LIN {X 0,Y 523.917,Z 120.846,A -85,B 0,C 180,E1 -4821.899,E2 -4821.899} C_VEL
LIN {X 0,Y 523.927,Z 120.846,A -85,B 0,C 180,E1 -4824.912,E2 -4824.912} C_VEL
LIN {X 0,Y 523.938,Z 120.844,A -85,B 0,C 180,E1 -4827.68,E2 -4827.68} C_VEL
LIN {X 0,Y 523.939,Z 120.843,A -85,B 0,C 180,E1 -4830.681,E2 -4830.681} C_VEL
LIN {X 0,Y 523.936,Z 120.839,A -85,B 0,C 180,E1 -4833.727,E2 -4833.727} C_VEL
LIN {X 0,Y 523.911,Z 120.845,A -85,B 0,C 180,E1 -4836.27,E2 -4836.27} C_VEL
LIN {X 0,Y 523.949,Z 120.845,A -85,B 0,C 180,E1 -4838.767,E2 -4838.767} C_VEL
LIN {X 0,Y 523.94,Z 120.843,A -85,B 0,C 180,E1 -4841.221,E2 -4841.221} C_VEL
LIN {X 0,Y 523.911,Z 120.843,A -85,B 0,C 180,E1 -4843.638,E2 -4843.638} C_VEL
LIN {X 0,Y 523.917,Z 120.845,A -85,B 0,C 180,E1 -4846.028,E2 -4846.028} C_VEL
LIN {X 0,Y 523.996,Z 120.835,A -85,B 0,C 180,E1 -4849.177,E2 -4849.177} C_VEL
LIN {X 0,Y 523.964,Z 120.844,A -85,B 0,C 180,E1 -4852.292,E2 -4852.292} C_VEL
LIN {X 0,Y 524.035,Z 120.834,A -85,B 0,C 180,E1 -4854.613,E2 -4854.613} C_VEL
LIN {X 0,Y 524.107,Z 120.819,A -85,B 0,C 180,E1 -4857.695,E2 -4857.695} C_VEL
LIN {X 0,Y 524.101,Z 120.817,A -85,B 0,C 180,E1 -4860,E2 -4860} C_VEL
LIN {X 0,Y 524.107,Z 120.825,A -85,B 0,C 180,E1 -4862.306,E2 -4862.306} C_VEL
LIN {X 0,Y 524.004,Z 120.837,A -85,B 0,C 180,E1 -4866.16,E2 -4866.16} C_VEL
LIN {X 0,Y 523.947,Z 120.832,A -85,B 0,C 180,E1 -4869.263,E2 -4869.263} C_VEL
LIN {X 0,Y 523.925,Z 120.843,A -85,B 0,C 180,E1 -4872.394,E2 -4872.394} C_VEL
LIN {X 0,Y 523.924,Z 120.843,A -85,B 0,C 180,E1 -4875.022,E2 -4875.022} C_VEL
LIN {X 0,Y 523.891,Z 120.851,A -85,B 0,C 180,E1 -4877.972,E2 -4877.972} C_VEL
LIN {X 0,Y 523.893,Z 120.847,A -85,B 0,C 180,E1 -4880.414,E2 -4880.414} C_VEL
LIN {X 0,Y 523.887,Z 120.847,A -85,B 0,C 180,E1 -4882.895,E2 -4882.895} C_VEL
LIN {X 0,Y 523.876,Z 120.857,A -85,B 0,C 180,E1 -4885.423,E2 -4885.423} C_VEL
LIN {X 0,Y 523.9,Z 120.841,A -85,B 0,C 180,E1 -4888.003,E2 -4888.003} C_VEL
LIN {X 0,Y 523.902,Z 120.842,A -85,B 0,C 180,E1 -4890.846,E2 -4890.846} C_VEL
LIN {X 0,Y 523.916,Z 120.846,A -85,B 0,C 180,E1 -4893.726,E2 -4893.726} C_VEL
LIN {X 0,Y 523.863,Z 120.849,A -85,B 0,C 180,E1 -4896.394,E2 -4896.394} C_VEL
LIN {X 0,Y 523.904,Z 120.848,A -85,B 0,C 180,E1 -4899.087,E2 -4899.087} C_VEL
LIN {X 0,Y 523.898,Z 120.847,A -85,B 0,C 180,E1 -4902.125,E2 -4902.125} C_VEL
LIN {X 0,Y 523.939,Z 120.837,A -85,B 0,C 180,E1 -4905.311,E2 -4905.311} C_VEL
LIN {X 0,Y 523.883,Z 120.852,A -85,B 0,C 180,E1 -4906.869,E2 -4906.869} C_VEL
LIN {X 0,Y 523.195,Z 120.935,A -85,B 0,C 180,E1 -4907.511,E2 -4907.511} C_VEL
LIN {X 0,Y 520.332,Z 121.296,A -85,B 0,C 180,E1 -4908.552,E2 -4908.552} C_VEL
LIN {X 0,Y 517.938,Z 121.591,A -85,B 0,C 180,E1 -4909.391,E2 -4909.391} C_VEL
LIN {X 0,Y 516.933,Z 121.716,A -85,B 0,C 180,E1 -4910.039,E2 -4910.039} C_VEL
LIN {X 0,Y 516.862,Z 121.727,A -85,B 0,C 180,E1 -4910.258,E2 -4910.258} C_VEL
LIN {X 0,Y 516.858,Z 121.723,A -85,B 0,C 180,E1 -4913.252,E2 -4913.252} C_VEL
LIN {X 0,Y 516.885,Z 121.724,A -85,B 0,C 180,E1 -4916.118,E2 -4916.118} C_VEL
LIN {X 0,Y 516.894,Z 121.721,A -85,B 0,C 180,E1 -4918.936,E2 -4918.936} C_VEL
LIN {X 0,Y 516.853,Z 121.724,A -85,B 0,C 180,E1 -4921.58,E2 -4921.58} C_VEL
LIN {X 0,Y 516.876,Z 121.73,A -85,B 0,C 180,E1 -4924.207,E2 -4924.207} C_VEL
LIN {X 0,Y 516.862,Z 121.725,A -85,B 0,C 180,E1 -4926.776,E2 -4926.776} C_VEL
LIN {X 0,Y 516.943,Z 121.718,A -85,B 0,C 180,E1 -4929.732,E2 -4929.732} C_VEL
LIN {X 0,Y 516.89,Z 121.718,A -85,B 0,C 180,E1 -4932.594,E2 -4932.594} C_VEL
LIN {X 0,Y 516.941,Z 121.714,A -85,B 0,C 180,E1 -4935.03,E2 -4935.03} C_VEL
LIN {X 0,Y 516.973,Z 121.714,A -85,B 0,C 180,E1 -4938.233,E2 -4938.233} C_VEL
LIN {X 0,Y 516.959,Z 121.718,A -85,B 0,C 180,E1 -4941.399,E2 -4941.399} C_VEL
LIN {X 0,Y 517.024,Z 121.796,A -85,B 0,C 180,E1 -4943.952,E2 -4943.952} C_VEL
LIN {X 0,Y 519.184,Z 132.355,A -85,B 0,C 180,E1 -4945.73,E2 -4945.73} C_VEL
LIN {X 0,Y 518.904,Z 142.438,A -85,B 0,C 180,E1 -4947.27,E2 -4947.27} C_VEL
LIN {X 0,Y 521.993,Z 156.093,A -85,B 0,C 180,E1 -4947.605,E2 -4947.605} C_VEL
LIN {X 0,Y 520.895,Z 307.149,A -85,B 0,C 180,E1 -4949.767,E2 -4949.767} C_VEL
LIN {X 0,Y 520.632,Z 322.808,A -85,B 0,C 180,E1 -4950.151,E2 -4950.151} C_VEL
LIN {X 0,Y 520.252,Z 336.624,A -85,B 0,C 180,E1 -4950.636,E2 -4950.636} C_VEL
LIN {X 0,Y 519.817,Z 350.651,A -85,B 0,C 180,E1 -4951.283,E2 -4951.283} C_VEL
LIN {X 0,Y 519.295,Z 363.702,A -85,B 0,C 180,E1 -4952.036,E2 -4952.036} C_VEL
LIN {X 0,Y 518.832,Z 376.141,A -85,B 0,C 180,E1 -4952.911,E2 -4952.911} C_VEL
LIN {X 0,Y 518.26,Z 388.801,A -85,B 0,C 180,E1 -4953.985,E2 -4953.985} C_VEL
LIN {X 0,Y 517.812,Z 399.431,A -85,B 0,C 180,E1 -4955.061,E2 -4955.061} C_VEL
LIN {X 0,Y 517.395,Z 409.318,A -85,B 0,C 180,E1 -4956.238,E2 -4956.238} C_VEL
LIN {X 0,Y 517.112,Z 418.47,A -85,B 0,C 180,E1 -4957.53,E2 -4957.53} C_VEL
LIN {X 0,Y 516.748,Z 427.144,A -85,B 0,C 180,E1 -4958.998,E2 -4958.998} C_VEL
LIN {X 0,Y 516.531,Z 434.772,A -85,B 0,C 180,E1 -4960.584,E2 -4960.584} C_VEL
LIN {X 0,Y 516.393,Z 440.872,A -85,B 0,C 180,E1 -4962.178,E2 -4962.178} C_VEL
LIN {X 0,Y 516.314,Z 445.566,A -85,B 0,C 180,E1 -4963.781,E2 -4963.781} C_VEL
LIN {X 0,Y 516.228,Z 448.212,A -85,B 0,C 180,E1 -4964.991,E2 -4964.991} C_VEL
LIN {X 0,Y 516.173,Z 450.688,A -85,B 0,C 180,E1 -4966.614,E2 -4966.614} C_VEL
LIN {X 0,Y 516.177,Z 451.931,A -85,B 0,C 180,E1 -4968.249,E2 -4968.249} C_VEL
LIN {X 0,Y 516.208,Z 451.919,A -85,B 0,C 180,E1 -4969.899,E2 -4969.899} C_VEL
LIN {X 0,Y 516.187,Z 450.606,A -85,B 0,C 180,E1 -4971.568,E2 -4971.568} C_VEL
LIN {X 0,Y 516.226,Z 447.945,A -85,B 0,C 180,E1 -4973.254,E2 -4973.254} C_VEL
LIN {X 0,Y 516.351,Z 443.836,A -85,B 0,C 180,E1 -4974.957,E2 -4974.957} C_VEL
LIN {X 0,Y 516.47,Z 438.125,A -85,B 0,C 180,E1 -4976.683,E2 -4976.683} C_VEL
LIN {X 0,Y 516.632,Z 432.137,A -85,B 0,C 180,E1 -4978.094,E2 -4978.094} C_VEL
LIN {X 0,Y 516.847,Z 424.84,A -85,B 0,C 180,E1 -4979.51,E2 -4979.51} C_VEL
LIN {X 0,Y 517.164,Z 416.46,A -85,B 0,C 180,E1 -4980.864,E2 -4980.864} C_VEL
LIN {X 0,Y 517.552,Z 406.602,A -85,B 0,C 180,E1 -4982.197,E2 -4982.197} C_VEL
LIN {X 0,Y 518.004,Z 395.547,A -85,B 0,C 180,E1 -4983.448,E2 -4983.448} C_VEL
LIN {X 0,Y 518.487,Z 383.913,A -85,B 0,C 180,E1 -4984.55,E2 -4984.55} C_VEL
LIN {X 0,Y 518.976,Z 372.041,A -85,B 0,C 180,E1 -4985.494,E2 -4985.494} C_VEL
LIN {X 0,Y 519.507,Z 359.348,A -85,B 0,C 180,E1 -4986.331,E2 -4986.331} C_VEL
LIN {X 0,Y 520.001,Z 344.499,A -85,B 0,C 180,E1 -4987.116,E2 -4987.116} C_VEL
LIN {X 0,Y 520.426,Z 329.396,A -85,B 0,C 180,E1 -4987.728,E2 -4987.728} C_VEL
LIN {X 0,Y 520.768,Z 314.128,A -85,B 0,C 180,E1 -4988.174,E2 -4988.174} C_VEL
LIN {X 0,Y 520.965,Z 298.076,A -85,B 0,C 180,E1 -4988.472,E2 -4988.472} C_VEL
LIN {X 0,Y 521.948,Z 155.747,A -85,B 0,C 180,E1 -4990.496,E2 -4990.496} C_VEL
LIN {X 0,Y 518.947,Z 142.396,A -85,B 0,C 180,E1 -4990.841,E2 -4990.841} C_VEL
LIN {X 0,Y 519.201,Z 132.665,A -85,B 0,C 180,E1 -4992.352,E2 -4992.352} C_VEL
LIN {X 0,Y 516.922,Z 121.722,A -85,B 0,C 180,E1 -4994.247,E2 -4994.247} C_VEL
LIN {X 0,Y 516.863,Z 121.729,A -85,B 0,C 180,E1 -4997.245,E2 -4997.245} C_VEL
LIN {X 0,Y 516.882,Z 121.726,A -85,B 0,C 180,E1 -4999.59,E2 -4999.59} C_VEL
LIN {X 0,Y 516.862,Z 121.73,A -85,B 0,C 180,E1 -5002.274,E2 -5002.274} C_VEL
LIN {X 0,Y 516.883,Z 121.718,A -85,B 0,C 180,E1 -5005.175,E2 -5005.175} C_VEL
LIN {X 0,Y 516.875,Z 121.725,A -85,B 0,C 180,E1 -5007.975,E2 -5007.975} C_VEL
LIN {X 0,Y 516.921,Z 121.716,A -85,B 0,C 180,E1 -5010.695,E2 -5010.695} C_VEL
LIN {X 0,Y 516.9,Z 121.724,A -85,B 0,C 180,E1 -5013.814,E2 -5013.814} C_VEL
LIN {X 0,Y 516.859,Z 121.722,A -85,B 0,C 180,E1 -5016.776,E2 -5016.776} C_VEL
LIN {X 0,Y 516.941,Z 121.719,A -85,B 0,C 180,E1 -5019.731,E2 -5019.731} C_VEL
LIN {X 0,Y 516.895,Z 121.719,A -85,B 0,C 180,E1 -5022.595,E2 -5022.595} C_VEL
LIN {X 0,Y 516.936,Z 121.713,A -85,B 0,C 180,E1 -5025.03,E2 -5025.03} C_VEL
LIN {X 0,Y 516.967,Z 121.711,A -85,B 0,C 180,E1 -5028.233,E2 -5028.233} C_VEL
LIN {X 0,Y 516.965,Z 121.715,A -85,B 0,C 180,E1 -5031.399,E2 -5031.399} C_VEL
LIN {X 0,Y 517.002,Z 121.709,A -85,B 0,C 180,E1 -5033.756,E2 -5033.756} C_VEL
LIN {X 0,Y 517.009,Z 121.707,A -85,B 0,C 180,E1 -5036.883,E2 -5036.883} C_VEL
LIN {X 0,Y 517.093,Z 121.699,A -85,B 0,C 180,E1 -5039.221,E2 -5039.221} C_VEL
LIN {X 0,Y 517.084,Z 121.694,A -85,B 0,C 180,E1 -5042.337,E2 -5042.337} C_VEL
LIN {X 0,Y 517.026,Z 121.708,A -85,B 0,C 180,E1 -5045.46,E2 -5045.46} C_VEL
LIN {X 0,Y 516.956,Z 121.712,A -85,B 0,C 180,E1 -5048.6,E2 -5048.6} C_VEL
LIN {X 0,Y 516.952,Z 121.711,A -85,B 0,C 180,E1 -5051.807,E2 -5051.807} C_VEL
LIN {X 0,Y 516.945,Z 121.717,A -85,B 0,C 180,E1 -5055.146,E2 -5055.146} C_VEL
LIN {X 0,Y 516.915,Z 121.717,A -85,B 0,C 180,E1 -5058.222,E2 -5058.222} C_VEL
LIN {X 0,Y 516.912,Z 121.721,A -85,B 0,C 180,E1 -5060.701,E2 -5060.701} C_VEL
LIN {X 0,Y 516.902,Z 121.718,A -85,B 0,C 180,E1 -5064.072,E2 -5064.072} C_VEL
LIN {X 0,Y 516.924,Z 121.721,A -85,B 0,C 180,E1 -5066.658,E2 -5066.658} C_VEL
LIN {X 0,Y 516.909,Z 121.716,A -85,B 0,C 180,E1 -5069.523,E2 -5069.523} C_VEL
LIN {X 0,Y 516.893,Z 121.725,A -85,B 0,C 180,E1 -5072.543,E2 -5072.543} C_VEL
LIN {X 0,Y 516.864,Z 121.723,A -85,B 0,C 180,E1 -5075.329,E2 -5075.329} C_VEL
LIN {X 0,Y 516.879,Z 121.722,A -85,B 0,C 180,E1 -5077.943,E2 -5077.943} C_VEL
LIN {X 0,Y 516.881,Z 121.725,A -85,B 0,C 180,E1 -5080.742,E2 -5080.742} C_VEL
LIN {X 0,Y 516.882,Z 121.718,A -85,B 0,C 180,E1 -5082.831,E2 -5082.831} C_VEL
LIN {X 0,Y 516.922,Z 121.717,A -85,B 0,C 180,E1 -5085.01,E2 -5085.01} C_VEL
LIN {X 0,Y 516.912,Z 121.723,A -85,B 0,C 180,E1 -5088.399,E2 -5088.399} C_VEL
LIN {X 0,Y 516.882,Z 121.723,A -85,B 0,C 180,E1 -5091.284,E2 -5091.284} C_VEL
LIN {X 0,Y 516.87,Z 121.728,A -85,B 0,C 180,E1 -5094.22,E2 -5094.22} C_VEL
LIN {X 0,Y 516.893,Z 121.719,A -85,B 0,C 180,E1 -5097.053,E2 -5097.053} C_VEL
LIN {X 0,Y 516.891,Z 121.728,A -85,B 0,C 180,E1 -5099.796,E2 -5099.796} C_VEL
LIN {X 0,Y 516.957,Z 121.813,A -85,B 0,C 180,E1 -5101.726,E2 -5101.726} C_VEL
LIN {X 0,Y 519.903,Z 134.937,A -85,B 0,C 180,E1 -5103.723,E2 -5103.723} C_VEL
LIN {X 0,Y 519.397,Z 152.164,A -85,B 0,C 180,E1 -5106.051,E2 -5106.051} C_VEL
LIN {X 0,Y 518.84,Z 168.384,A -85,B 0,C 180,E1 -5108.2,E2 -5108.2} C_VEL
LIN {X 0,Y 521.885,Z 184.442,A -85,B 0,C 180,E1 -5108.571,E2 -5108.571} C_VEL
LIN {X 0,Y 520.825,Z 334.017,A -85,B 0,C 180,E1 -5110.708,E2 -5110.708} C_VEL
LIN {X 0,Y 520.462,Z 349.322,A -85,B 0,C 180,E1 -5111.07,E2 -5111.07} C_VEL
LIN {X 0,Y 520.092,Z 364.284,A -85,B 0,C 180,E1 -5111.587,E2 -5111.587} C_VEL
LIN {X 0,Y 519.608,Z 377.4,A -85,B 0,C 180,E1 -5112.181,E2 -5112.181} C_VEL
LIN {X 0,Y 519.123,Z 391.385,A -85,B 0,C 180,E1 -5112.977,E2 -5112.977} C_VEL
LIN {X 0,Y 518.608,Z 404.708,A -85,B 0,C 180,E1 -5113.911,E2 -5113.911} C_VEL
LIN {X 0,Y 518.103,Z 416.289,A -85,B 0,C 180,E1 -5114.886,E2 -5114.886} C_VEL
LIN {X 0,Y 517.642,Z 427.963,A -85,B 0,C 180,E1 -5116.055,E2 -5116.055} C_VEL
LIN {X 0,Y 517.25,Z 437.985,A -85,B 0,C 180,E1 -5117.245,E2 -5117.245} C_VEL
LIN {X 0,Y 516.899,Z 447.853,A -85,B 0,C 180,E1 -5118.64,E2 -5118.64} C_VEL
LIN {X 0,Y 516.662,Z 455.969,A -85,B 0,C 180,E1 -5120.013,E2 -5120.013} C_VEL
LIN {X 0,Y 516.513,Z 462.728,A -85,B 0,C 180,E1 -5121.392,E2 -5121.392} C_VEL
LIN {X 0,Y 516.39,Z 468.972,A -85,B 0,C 180,E1 -5122.965,E2 -5122.965} C_VEL
LIN {X 0,Y 516.352,Z 473.803,A -85,B 0,C 180,E1 -5124.533,E2 -5124.533} C_VEL
LIN {X 0,Y 516.277,Z 477.339,A -85,B 0,C 180,E1 -5126.097,E2 -5126.097} C_VEL
LIN {X 0,Y 516.258,Z 479.667,A -85,B 0,C 180,E1 -5127.66,E2 -5127.66} C_VEL
LIN {X 0,Y 516.156,Z 480.837,A -85,B 0,C 180,E1 -5129.22,E2 -5129.22} C_VEL
LIN {X 0,Y 516.156,Z 480.838,A -85,B 0,C 180,E1 -5130.78,E2 -5130.78} C_VEL
LIN {X 0,Y 516.258,Z 479.668,A -85,B 0,C 180,E1 -5132.341,E2 -5132.341} C_VEL
LIN {X 0,Y 516.277,Z 477.344,A -85,B 0,C 180,E1 -5133.903,E2 -5133.903} C_VEL
LIN {X 0,Y 516.353,Z 473.817,A -85,B 0,C 180,E1 -5135.468,E2 -5135.468} C_VEL
LIN {X 0,Y 516.395,Z 468.994,A -85,B 0,C 180,E1 -5137.036,E2 -5137.036} C_VEL
LIN {X 0,Y 516.513,Z 462.748,A -85,B 0,C 180,E1 -5138.608,E2 -5138.608} C_VEL
LIN {X 0,Y 516.747,Z 454.903,A -85,B 0,C 180,E1 -5140.184,E2 -5140.184} C_VEL
LIN {X 0,Y 516.964,Z 446.558,A -85,B 0,C 180,E1 -5141.568,E2 -5141.568} C_VEL
LIN {X 0,Y 517.312,Z 436.503,A -85,B 0,C 180,E1 -5142.954,E2 -5142.954} C_VEL
LIN {X 0,Y 517.713,Z 426.224,A -85,B 0,C 180,E1 -5144.144,E2 -5144.144} C_VEL
LIN {X 0,Y 518.203,Z 414.493,A -85,B 0,C 180,E1 -5145.287,E2 -5145.287} C_VEL
LIN {X 0,Y 518.702,Z 401.673,A -85,B 0,C 180,E1 -5146.329,E2 -5146.329} C_VEL
LIN {X 0,Y 519.287,Z 388.287,A -85,B 0,C 180,E1 -5147.221,E2 -5147.221} C_VEL
LIN {X 0,Y 519.715,Z 375.496,A -85,B 0,C 180,E1 -5147.918,E2 -5147.918} C_VEL
LIN {X 0,Y 520.196,Z 360.49,A -85,B 0,C 180,E1 -5148.563,E2 -5148.563} C_VEL
LIN {X 0,Y 520.557,Z 345.891,A -85,B 0,C 180,E1 -5149.027,E2 -5149.027} C_VEL
LIN {X 0,Y 520.827,Z 330.839,A -85,B 0,C 180,E1 -5149.349,E2 -5149.349} C_VEL
LIN {X 0,Y 521.892,Z 184.236,A -85,B 0,C 180,E1 -5151.433,E2 -5151.433} C_VEL
LIN {X 0,Y 518.848,Z 168.523,A -85,B 0,C 180,E1 -5151.799,E2 -5151.799} C_VEL
LIN {X 0,Y 519.589,Z 147.552,A -85,B 0,C 180,E1 -5154.578,E2 -5154.578} C_VEL
LIN {X 0,Y 519.965,Z 134.961,A -85,B 0,C 180,E1 -5156.274,E2 -5156.274} C_VEL
LIN {X 0,Y 516.919,Z 121.724,A -85,B 0,C 180,E1 -5158.276,E2 -5158.276} C_VEL
LIN {X 0,Y 516.891,Z 121.722,A -85,B 0,C 180,E1 -5161.11,E2 -5161.11} C_VEL
LIN {X 0,Y 516.91,Z 121.726,A -85,B 0,C 180,E1 -5163.966,E2 -5163.966} C_VEL
LIN {X 0,Y 516.878,Z 121.724,A -85,B 0,C 180,E1 -5166.747,E2 -5166.747} C_VEL
LIN {X 0,Y 516.885,Z 121.729,A -85,B 0,C 180,E1 -5169.722,E2 -5169.722} C_VEL
LIN {X 0,Y 516.909,Z 121.726,A -85,B 0,C 180,E1 -5171.776,E2 -5171.776} C_VEL
LIN {X 0,Y 516.897,Z 121.722,A -85,B 0,C 180,E1 -5175.007,E2 -5175.007} C_VEL
LIN {X 0,Y 516.916,Z 121.718,A -85,B 0,C 180,E1 -5178.399,E2 -5178.399} C_VEL
LIN {X 0,Y 516.88,Z 121.725,A -85,B 0,C 180,E1 -5181.284,E2 -5181.284} C_VEL
LIN {X 0,Y 516.874,Z 121.721,A -85,B 0,C 180,E1 -5184.22,E2 -5184.22} C_VEL
LIN {X 0,Y 516.884,Z 121.726,A -85,B 0,C 180,E1 -5187.052,E2 -5187.052} C_VEL
LIN {X 0,Y 516.87,Z 121.722,A -85,B 0,C 180,E1 -5189.795,E2 -5189.795} C_VEL
LIN {X 0,Y 516.886,Z 121.714,A -85,B 0,C 180,E1 -5192.465,E2 -5192.465} C_VEL
LIN {X 0,Y 516.852,Z 121.731,A -85,B 0,C 180,E1 -5195.069,E2 -5195.069} C_VEL
LIN {X 0,Y 516.873,Z 121.72,A -85,B 0,C 180,E1 -5197.622,E2 -5197.622} C_VEL
LIN {X 0,Y 516.933,Z 121.714,A -85,B 0,C 180,E1 -5200.13,E2 -5200.13} C_VEL
LIN {X 0,Y 516.897,Z 121.724,A -85,B 0,C 180,E1 -5202.595,E2 -5202.595} C_VEL
LIN {X 0,Y 516.936,Z 121.718,A -85,B 0,C 180,E1 -5205.03,E2 -5205.03} C_VEL
LIN {X 0,Y 516.972,Z 121.711,A -85,B 0,C 180,E1 -5208.234,E2 -5208.234} C_VEL
LIN {X 0,Y 516.955,Z 121.71,A -85,B 0,C 180,E1 -5211.4,E2 -5211.4} C_VEL
LIN {X 0,Y 516.986,Z 121.714,A -85,B 0,C 180,E1 -5214.54,E2 -5214.54} C_VEL
LIN {X 0,Y 517.077,Z 121.694,A -85,B 0,C 180,E1 -5217.663,E2 -5217.663} C_VEL
LIN {X 0,Y 517.069,Z 121.692,A -85,B 0,C 180,E1 -5220,E2 -5220} C_VEL
LIN {X 0,Y 517.077,Z 121.701,A -85,B 0,C 180,E1 -5222.337,E2 -5222.337} C_VEL
LIN {X 0,Y 516.971,Z 121.711,A -85,B 0,C 180,E1 -5226.244,E2 -5226.244} C_VEL
LIN {X 0,Y 516.909,Z 121.709,A -85,B 0,C 180,E1 -5229.39,E2 -5229.39} C_VEL
LIN {X 0,Y 516.885,Z 121.719,A -85,B 0,C 180,E1 -5232.566,E2 -5232.566} C_VEL
LIN {X 0,Y 516.889,Z 121.721,A -85,B 0,C 180,E1 -5235.121,E2 -5235.121} C_VEL
LIN {X 0,Y 516.84,Z 121.726,A -85,B 0,C 180,E1 -5238.226,E2 -5238.226} C_VEL
LIN {X 0,Y 516.859,Z 121.723,A -85,B 0,C 180,E1 -5240.704,E2 -5240.704} C_VEL
LIN {X 0,Y 516.841,Z 121.729,A -85,B 0,C 180,E1 -5243.225,E2 -5243.225} C_VEL
LIN {X 0,Y 516.861,Z 121.722,A -85,B 0,C 180,E1 -5246.176,E2 -5246.176} C_VEL
LIN {X 0,Y 516.833,Z 121.72,A -85,B 0,C 180,E1 -5248.421,E2 -5248.421} C_VEL
LIN {X 0,Y 516.853,Z 121.724,A -85,B 0,C 180,E1 -5251.112,E2 -5251.112} C_VEL
LIN {X 0,Y 516.874,Z 121.721,A -85,B 0,C 180,E1 -5253.959,E2 -5253.959} C_VEL
LIN {X 0,Y 516.812,Z 121.731,A -85,B 0,C 180,E1 -5256.752,E2 -5256.752} C_VEL
LIN {X 0,Y 516.86,Z 121.72,A -85,B 0,C 180,E1 -5259.724,E2 -5259.724} C_VEL
LIN {X 0,Y 516.847,Z 121.733,A -85,B 0,C 180,E1 -5262.836,E2 -5262.836} C_VEL
LIN {X 0,Y 516.901,Z 121.717,A -85,B 0,C 180,E1 -5265.007,E2 -5265.007} C_VEL
LIN {X 0,Y 516.854,Z 121.727,A -85,B 0,C 180,E1 -5268.407,E2 -5268.407} C_VEL
LIN {X 0,Y 516.862,Z 121.727,A -85,B 0,C 180,E1 -5270.258,E2 -5270.258} C_VEL
LIN {X 0,Y 516.225,Z 121.811,A -85,B 0,C 180,E1 -5270.908,E2 -5270.908} C_VEL
LIN {X 0,Y 513.381,Z 122.162,A -85,B 0,C 180,E1 -5271.964,E2 -5271.964} C_VEL
LIN {X 0,Y 510.953,Z 122.462,A -85,B 0,C 180,E1 -5272.814,E2 -5272.814} C_VEL
LIN {X 0,Y 509.901,Z 122.589,A -85,B 0,C 180,E1 -5273.471,E2 -5273.471} C_VEL
LIN {X 0,Y 509.812,Z 122.6,A -85,B 0,C 180,E1 -5273.693,E2 -5273.693} C_VEL
LIN {X 0,Y 509.844,Z 122.6,A -85,B 0,C 180,E1 -5276.537,E2 -5276.537} C_VEL
LIN {X 0,Y 509.84,Z 122.599,A -85,B 0,C 180,E1 -5279.333,E2 -5279.333} C_VEL
LIN {X 0,Y 509.838,Z 122.602,A -85,B 0,C 180,E1 -5282.051,E2 -5282.051} C_VEL
LIN {X 0,Y 509.807,Z 122.605,A -85,B 0,C 180,E1 -5284.7,E2 -5284.7} C_VEL
LIN {X 0,Y 509.831,Z 122.601,A -85,B 0,C 180,E1 -5287.458,E2 -5287.458} C_VEL
LIN {X 0,Y 509.921,Z 122.594,A -85,B 0,C 180,E1 -5289.844,E2 -5289.844} C_VEL
LIN {X 0,Y 509.861,Z 122.593,A -85,B 0,C 180,E1 -5293.174,E2 -5293.174} C_VEL
LIN {X 0,Y 509.86,Z 122.6,A -85,B 0,C 180,E1 -5295.634,E2 -5295.634} C_VEL
LIN {X 0,Y 509.917,Z 122.591,A -85,B 0,C 180,E1 -5298.874,E2 -5298.874} C_VEL
LIN {X 0,Y 509.914,Z 122.595,A -85,B 0,C 180,E1 -5302.078,E2 -5302.078} C_VEL
LIN {X 0,Y 509.985,Z 122.776,A -85,B 0,C 180,E1 -5303.72,E2 -5303.72} C_VEL
LIN {X 0,Y 512.348,Z 134.221,A -85,B 0,C 180,E1 -5305.673,E2 -5305.673} C_VEL
LIN {X 0,Y 512.067,Z 142.424,A -85,B 0,C 180,E1 -5306.95,E2 -5306.95} C_VEL
LIN {X 0,Y 515.384,Z 157.14,A -85,B 0,C 180,E1 -5307.332,E2 -5307.332} C_VEL
LIN {X 0,Y 514.206,Z 307.466,A -85,B 0,C 180,E1 -5309.51,E2 -5309.51} C_VEL
LIN {X 0,Y 513.917,Z 323.162,A -85,B 0,C 180,E1 -5309.902,E2 -5309.902} C_VEL
LIN {X 0,Y 513.443,Z 338.552,A -85,B 0,C 180,E1 -5310.458,E2 -5310.458} C_VEL
LIN {X 0,Y 512.956,Z 353.375,A -85,B 0,C 180,E1 -5311.177,E2 -5311.177} C_VEL
LIN {X 0,Y 512.4,Z 366.385,A -85,B 0,C 180,E1 -5311.965,E2 -5311.965} C_VEL
LIN {X 0,Y 511.851,Z 379.638,A -85,B 0,C 180,E1 -5312.951,E2 -5312.951} C_VEL
LIN {X 0,Y 511.246,Z 391.752,A -85,B 0,C 180,E1 -5314.04,E2 -5314.04} C_VEL
LIN {X 0,Y 510.737,Z 403.655,A -85,B 0,C 180,E1 -5315.329,E2 -5315.329} C_VEL
LIN {X 0,Y 510.292,Z 414.317,A -85,B 0,C 180,E1 -5316.723,E2 -5316.723} C_VEL
LIN {X 0,Y 509.902,Z 423.246,A -85,B 0,C 180,E1 -5318.121,E2 -5318.121} C_VEL
LIN {X 0,Y 509.625,Z 430.68,A -85,B 0,C 180,E1 -5319.525,E2 -5319.525} C_VEL
LIN {X 0,Y 509.416,Z 437.657,A -85,B 0,C 180,E1 -5321.136,E2 -5321.136} C_VEL
LIN {X 0,Y 509.261,Z 443.16,A -85,B 0,C 180,E1 -5322.756,E2 -5322.756} C_VEL
LIN {X 0,Y 509.17,Z 447.306,A -85,B 0,C 180,E1 -5324.386,E2 -5324.386} C_VEL
LIN {X 0,Y 509.061,Z 450.186,A -85,B 0,C 180,E1 -5326.028,E2 -5326.028} C_VEL
LIN {X 0,Y 509.096,Z 451.849,A -85,B 0,C 180,E1 -5327.722,E2 -5327.722} C_VEL
LIN {X 0,Y 509.075,Z 452.232,A -85,B 0,C 180,E1 -5329.349,E2 -5329.349} C_VEL
LIN {X 0,Y 509.072,Z 451.373,A -85,B 0,C 180,E1 -5331.035,E2 -5331.035} C_VEL
LIN {X 0,Y 509.121,Z 449.189,A -85,B 0,C 180,E1 -5332.738,E2 -5332.738} C_VEL
LIN {X 0,Y 509.261,Z 445.583,A -85,B 0,C 180,E1 -5334.457,E2 -5334.457} C_VEL
LIN {X 0,Y 509.361,Z 440.409,A -85,B 0,C 180,E1 -5336.201,E2 -5336.201} C_VEL
LIN {X 0,Y 509.49,Z 435.406,A -85,B 0,C 180,E1 -5337.523,E2 -5337.523} C_VEL
LIN {X 0,Y 509.71,Z 428.176,A -85,B 0,C 180,E1 -5339.074,E2 -5339.074} C_VEL
LIN {X 0,Y 510.014,Z 420.521,A -85,B 0,C 180,E1 -5340.425,E2 -5340.425} C_VEL
LIN {X 0,Y 510.401,Z 411.372,A -85,B 0,C 180,E1 -5341.782,E2 -5341.782} C_VEL
LIN {X 0,Y 510.884,Z 400.607,A -85,B 0,C 180,E1 -5343.116,E2 -5343.116} C_VEL
LIN {X 0,Y 511.374,Z 389.209,A -85,B 0,C 180,E1 -5344.296,E2 -5344.296} C_VEL
LIN {X 0,Y 511.923,Z 377.32,A -85,B 0,C 180,E1 -5345.327,E2 -5345.327} C_VEL
LIN {X 0,Y 512.486,Z 364.431,A -85,B 0,C 180,E1 -5346.256,E2 -5346.256} C_VEL
LIN {X 0,Y 513.071,Z 350.613,A -85,B 0,C 180,E1 -5347.064,E2 -5347.064} C_VEL
LIN {X 0,Y 513.505,Z 336.531,A -85,B 0,C 180,E1 -5347.718,E2 -5347.718} C_VEL
LIN {X 0,Y 513.89,Z 321.316,A -85,B 0,C 180,E1 -5348.247,E2 -5348.247} C_VEL
LIN {X 0,Y 514.203,Z 305.959,A -85,B 0,C 180,E1 -5348.61,E2 -5348.61} C_VEL
LIN {X 0,Y 515.413,Z 157.087,A -85,B 0,C 180,E1 -5350.77,E2 -5350.77} C_VEL
LIN {X 0,Y 512.147,Z 142.534,A -85,B 0,C 180,E1 -5351.164,E2 -5351.164} C_VEL
LIN {X 0,Y 512.329,Z 134.01,A -85,B 0,C 180,E1 -5352.508,E2 -5352.508} C_VEL
LIN {X 0,Y 509.865,Z 122.603,A -85,B 0,C 180,E1 -5354.508,E2 -5354.508} C_VEL
LIN {X 0,Y 509.817,Z 122.606,A -85,B 0,C 180,E1 -5357.508,E2 -5357.508} C_VEL
LIN {X 0,Y 509.843,Z 122.607,A -85,B 0,C 180,E1 -5360.647,E2 -5360.647} C_VEL
LIN {X 0,Y 509.811,Z 122.605,A -85,B 0,C 180,E1 -5363.645,E2 -5363.645} C_VEL
LIN {X 0,Y 509.86,Z 122.6,A -85,B 0,C 180,E1 -5366.539,E2 -5366.539} C_VEL
LIN {X 0,Y 509.843,Z 122.598,A -85,B 0,C 180,E1 -5369.334,E2 -5369.334} C_VEL
LIN {X 0,Y 509.851,Z 122.598,A -85,B 0,C 180,E1 -5372.052,E2 -5372.052} C_VEL
LIN {X 0,Y 509.81,Z 122.601,A -85,B 0,C 180,E1 -5374.7,E2 -5374.7} C_VEL
LIN {X 0,Y 509.827,Z 122.6,A -85,B 0,C 180,E1 -5377.458,E2 -5377.458} C_VEL
LIN {X 0,Y 509.917,Z 122.594,A -85,B 0,C 180,E1 -5379.844,E2 -5379.844} C_VEL
LIN {X 0,Y 509.863,Z 122.596,A -85,B 0,C 180,E1 -5383.174,E2 -5383.174} C_VEL
LIN {X 0,Y 509.856,Z 122.601,A -85,B 0,C 180,E1 -5385.633,E2 -5385.633} C_VEL
LIN {X 0,Y 509.914,Z 122.588,A -85,B 0,C 180,E1 -5388.874,E2 -5388.874} C_VEL
LIN {X 0,Y 509.952,Z 122.587,A -85,B 0,C 180,E1 -5392.078,E2 -5392.078} C_VEL
LIN {X 0,Y 509.978,Z 122.578,A -85,B 0,C 180,E1 -5394.464,E2 -5394.464} C_VEL
LIN {X 0,Y 510.056,Z 122.574,A -85,B 0,C 180,E1 -5397.631,E2 -5397.631} C_VEL
LIN {X 0,Y 510.062,Z 122.572,A -85,B 0,C 180,E1 -5400.789,E2 -5400.789} C_VEL
LIN {X 0,Y 509.952,Z 122.589,A -85,B 0,C 180,E1 -5403.16,E2 -5403.16} C_VEL
LIN {X 0,Y 509.942,Z 122.585,A -85,B 0,C 180,E1 -5406.33,E2 -5406.33} C_VEL
LIN {X 0,Y 509.904,Z 122.592,A -85,B 0,C 180,E1 -5408.72,E2 -5408.72} C_VEL
LIN {X 0,Y 509.905,Z 122.588,A -85,B 0,C 180,E1 -5411.931,E2 -5411.931} C_VEL
LIN {X 0,Y 509.894,Z 122.594,A -85,B 0,C 180,E1 -5415.242,E2 -5415.242} C_VEL
LIN {X 0,Y 509.86,Z 122.598,A -85,B 0,C 180,E1 -5418.483,E2 -5418.483} C_VEL
LIN {X 0,Y 509.85,Z 122.603,A -85,B 0,C 180,E1 -5421.001,E2 -5421.001} C_VEL
LIN {X 0,Y 509.864,Z 122.598,A -85,B 0,C 180,E1 -5424.426,E2 -5424.426} C_VEL
LIN {X 0,Y 509.883,Z 122.597,A -85,B 0,C 180,E1 -5427.056,E2 -5427.056} C_VEL
LIN {X 0,Y 509.856,Z 122.595,A -85,B 0,C 180,E1 -5429.751,E2 -5429.751} C_VEL
LIN {X 0,Y 509.866,Z 122.601,A -85,B 0,C 180,E1 -5432.773,E2 -5432.773} C_VEL
LIN {X 0,Y 509.824,Z 122.6,A -85,B 0,C 180,E1 -5435.578,E2 -5435.578} C_VEL
LIN {X 0,Y 509.848,Z 122.597,A -85,B 0,C 180,E1 -5438.338,E2 -5438.338} C_VEL
LIN {X 0,Y 509.854,Z 122.597,A -85,B 0,C 180,E1 -5441.425,E2 -5441.425} C_VEL
LIN {X 0,Y 509.856,Z 122.6,A -85,B 0,C 180,E1 -5444.668,E2 -5444.668} C_VEL
LIN {X 0,Y 509.854,Z 122.602,A -85,B 0,C 180,E1 -5448.103,E2 -5448.103} C_VEL
LIN {X 0,Y 509.846,Z 122.601,A -85,B 0,C 180,E1 -5450.648,E2 -5450.648} C_VEL
LIN {X 0,Y 509.823,Z 122.604,A -85,B 0,C 180,E1 -5453.647,E2 -5453.647} C_VEL
LIN {X 0,Y 509.858,Z 122.598,A -85,B 0,C 180,E1 -5456.539,E2 -5456.539} C_VEL
LIN {X 0,Y 509.844,Z 122.602,A -85,B 0,C 180,E1 -5459.334,E2 -5459.334} C_VEL
LIN {X 0,Y 509.899,Z 122.765,A -85,B 0,C 180,E1 -5461.445,E2 -5461.445} C_VEL
LIN {X 0,Y 513.046,Z 136.393,A -85,B 0,C 180,E1 -5463.564,E2 -5463.564} C_VEL
LIN {X 0,Y 512.647,Z 150.454,A -85,B 0,C 180,E1 -5465.5,E2 -5465.5} C_VEL
LIN {X 0,Y 511.982,Z 168.119,A -85,B 0,C 180,E1 -5467.88,E2 -5467.88} C_VEL
LIN {X 0,Y 515.302,Z 185.498,A -85,B 0,C 180,E1 -5468.298,E2 -5468.298} C_VEL
LIN {X 0,Y 514.112,Z 334.502,A -85,B 0,C 180,E1 -5470.459,E2 -5470.459} C_VEL
LIN {X 0,Y 513.737,Z 350.334,A -85,B 0,C 180,E1 -5470.85,E2 -5470.85} C_VEL
LIN {X 0,Y 513.303,Z 365.436,A -85,B 0,C 180,E1 -5471.393,E2 -5471.393} C_VEL
LIN {X 0,Y 512.773,Z 379.142,A -85,B 0,C 180,E1 -5472.039,E2 -5472.039} C_VEL
LIN {X 0,Y 512.206,Z 392.728,A -85,B 0,C 180,E1 -5472.843,E2 -5472.843} C_VEL
LIN {X 0,Y 511.636,Z 406.547,A -85,B 0,C 180,E1 -5473.85,E2 -5473.85} C_VEL
LIN {X 0,Y 511.04,Z 419.048,A -85,B 0,C 180,E1 -5474.955,E2 -5474.955} C_VEL
LIN {X 0,Y 510.532,Z 431.312,A -85,B 0,C 180,E1 -5476.263,E2 -5476.263} C_VEL
LIN {X 0,Y 510.079,Z 442.209,A -85,B 0,C 180,E1 -5477.669,E2 -5477.669} C_VEL
LIN {X 0,Y 509.8,Z 451.283,A -85,B 0,C 180,E1 -5479.073,E2 -5479.073} C_VEL
LIN {X 0,Y 509.498,Z 458.805,A -85,B 0,C 180,E1 -5480.472,E2 -5480.472} C_VEL
LIN {X 0,Y 509.356,Z 465.828,A -85,B 0,C 180,E1 -5482.069,E2 -5482.069} C_VEL
LIN {X 0,Y 509.264,Z 471.349,A -85,B 0,C 180,E1 -5483.662,E2 -5483.662} C_VEL
LIN {X 0,Y 509.157,Z 475.522,A -85,B 0,C 180,E1 -5485.25,E2 -5485.25} C_VEL
LIN {X 0,Y 509.185,Z 478.45,A -85,B 0,C 180,E1 -5486.835,E2 -5486.835} C_VEL
LIN {X 0,Y 509.109,Z 480.194,A -85,B 0,C 180,E1 -5488.418,E2 -5488.418} C_VEL
LIN {X 0,Y 509.063,Z 480.794,A -85,B 0,C 180,E1 -5490,E2 -5490} C_VEL
LIN {X 0,Y 509.11,Z 480.197,A -85,B 0,C 180,E1 -5491.582,E2 -5491.582} C_VEL
LIN {X 0,Y 509.185,Z 478.455,A -85,B 0,C 180,E1 -5493.165,E2 -5493.165} C_VEL
LIN {X 0,Y 509.157,Z 475.535,A -85,B 0,C 180,E1 -5494.751,E2 -5494.751} C_VEL
LIN {X 0,Y 509.286,Z 471.375,A -85,B 0,C 180,E1 -5496.339,E2 -5496.339} C_VEL
LIN {X 0,Y 509.356,Z 465.856,A -85,B 0,C 180,E1 -5497.931,E2 -5497.931} C_VEL
LIN {X 0,Y 509.499,Z 458.834,A -85,B 0,C 180,E1 -5499.528,E2 -5499.528} C_VEL
LIN {X 0,Y 509.818,Z 451.323,A -85,B 0,C 180,E1 -5500.927,E2 -5500.927} C_VEL
LIN {X 0,Y 510.074,Z 442.263,A -85,B 0,C 180,E1 -5502.332,E2 -5502.332} C_VEL
LIN {X 0,Y 510.534,Z 431.375,A -85,B 0,C 180,E1 -5503.737,E2 -5503.737} C_VEL
LIN {X 0,Y 511.054,Z 419.129,A -85,B 0,C 180,E1 -5505.045,E2 -5505.045} C_VEL
LIN {X 0,Y 511.635,Z 406.643,A -85,B 0,C 180,E1 -5506.151,E2 -5506.151} C_VEL
LIN {X 0,Y 512.146,Z 394.367,A -85,B 0,C 180,E1 -5507.057,E2 -5507.057} C_VEL
LIN {X 0,Y 512.688,Z 381.091,A -85,B 0,C 180,E1 -5507.862,E2 -5507.862} C_VEL
LIN {X 0,Y 513.25,Z 366.643,A -85,B 0,C 180,E1 -5508.561,E2 -5508.561} C_VEL
LIN {X 0,Y 513.705,Z 351.443,A -85,B 0,C 180,E1 -5509.119,E2 -5509.119} C_VEL
LIN {X 0,Y 514.047,Z 336.346,A -85,B 0,C 180,E1 -5509.506,E2 -5509.506} C_VEL
LIN {X 0,Y 514.324,Z 305.655,A -85,B 0,C 180,E1 -5509.976,E2 -5509.976} C_VEL
LIN {X 0,Y 515.284,Z 185.159,A -85,B 0,C 180,E1 -5511.703,E2 -5511.703} C_VEL
LIN {X 0,Y 511.975,Z 168.304,A -85,B 0,C 180,E1 -5512.107,E2 -5512.107} C_VEL
LIN {X 0,Y 512.725,Z 148.907,A -85,B 0,C 180,E1 -5514.713,E2 -5514.713} C_VEL
LIN {X 0,Y 513.057,Z 136.309,A -85,B 0,C 180,E1 -5516.436,E2 -5516.436} C_VEL
LIN {X 0,Y 509.883,Z 122.598,A -85,B 0,C 180,E1 -5518.551,E2 -5518.551} C_VEL
LIN {X 0,Y 509.822,Z 122.605,A -85,B 0,C 180,E1 -5521.591,E2 -5521.591} C_VEL
LIN {X 0,Y 509.849,Z 122.603,A -85,B 0,C 180,E1 -5524.414,E2 -5524.414} C_VEL
LIN {X 0,Y 509.819,Z 122.605,A -85,B 0,C 180,E1 -5527.341,E2 -5527.341} C_VEL
LIN {X 0,Y 509.84,Z 122.6,A -85,B 0,C 180,E1 -5530.383,E2 -5530.383} C_VEL
LIN {X 0,Y 509.806,Z 122.604,A -85,B 0,C 180,E1 -5533.06,E2 -5533.06} C_VEL
LIN {X 0,Y 509.825,Z 122.607,A -85,B 0,C 180,E1 -5535.794,E2 -5535.794} C_VEL
LIN {X 0,Y 509.858,Z 122.597,A -85,B 0,C 180,E1 -5538.575,E2 -5538.575} C_VEL
LIN {X 0,Y 509.852,Z 122.599,A -85,B 0,C 180,E1 -5541.787,E2 -5541.787} C_VEL
LIN {X 0,Y 509.832,Z 122.599,A -85,B 0,C 180,E1 -5544.622,E2 -5544.622} C_VEL
LIN {X 0,Y 509.863,Z 122.6,A -85,B 0,C 180,E1 -5547.481,E2 -5547.481} C_VEL
LIN {X 0,Y 509.856,Z 122.595,A -85,B 0,C 180,E1 -5550.275,E2 -5550.275} C_VEL
LIN {X 0,Y 509.879,Z 122.591,A -85,B 0,C 180,E1 -5553.63,E2 -5553.63} C_VEL
LIN {X 0,Y 509.821,Z 122.602,A -85,B 0,C 180,E1 -5556.436,E2 -5556.436} C_VEL
LIN {X 0,Y 509.919,Z 122.587,A -85,B 0,C 180,E1 -5559.845,E2 -5559.845} C_VEL
LIN {X 0,Y 509.861,Z 122.596,A -85,B 0,C 180,E1 -5563.174,E2 -5563.174} C_VEL
LIN {X 0,Y 509.849,Z 122.597,A -85,B 0,C 180,E1 -5565.634,E2 -5565.634} C_VEL
LIN {X 0,Y 509.916,Z 122.592,A -85,B 0,C 180,E1 -5568.875,E2 -5568.875} C_VEL
LIN {X 0,Y 509.889,Z 122.594,A -85,B 0,C 180,E1 -5572.078,E2 -5572.078} C_VEL
LIN {X 0,Y 509.941,Z 122.592,A -85,B 0,C 180,E1 -5574.464,E2 -5574.464} C_VEL
LIN {X 0,Y 510.045,Z 122.57,A -85,B 0,C 180,E1 -5577.631,E2 -5577.631} C_VEL
LIN {X 0,Y 510.038,Z 122.567,A -85,B 0,C 180,E1 -5580,E2 -5580} C_VEL
LIN {X 0,Y 510.045,Z 122.576,A -85,B 0,C 180,E1 -5582.369,E2 -5582.369} C_VEL
LIN {X 0,Y 509.938,Z 122.587,A -85,B 0,C 180,E1 -5585.537,E2 -5585.537} C_VEL
LIN {X 0,Y 509.879,Z 122.592,A -85,B 0,C 180,E1 -5587.923,E2 -5587.923} C_VEL
LIN {X 0,Y 509.865,Z 122.588,A -85,B 0,C 180,E1 -5591.127,E2 -5591.127} C_VEL
LIN {X 0,Y 509.821,Z 122.604,A -85,B 0,C 180,E1 -5593.554,E2 -5593.554} C_VEL
LIN {X 0,Y 509.793,Z 122.605,A -85,B 0,C 180,E1 -5596.005,E2 -5596.005} C_VEL
LIN {X 0,Y 509.806,Z 122.601,A -85,B 0,C 180,E1 -5598.486,E2 -5598.486} C_VEL
LIN {X 0,Y 509.812,Z 122.603,A -85,B 0,C 180,E1 -5601.004,E2 -5601.004} C_VEL
LIN {X 0,Y 509.802,Z 122.61,A -85,B 0,C 180,E1 -5603.565,E2 -5603.565} C_VEL
LIN {X 0,Y 509.802,Z 122.601,A -85,B 0,C 180,E1 -5606.352,E2 -5606.352} C_VEL
LIN {X 0,Y 509.797,Z 122.599,A -85,B 0,C 180,E1 -5608.85,E2 -5608.85} C_VEL
LIN {X 0,Y 509.792,Z 122.605,A -85,B 0,C 180,E1 -5611.593,E2 -5611.593} C_VEL
LIN {X 0,Y 509.832,Z 122.599,A -85,B 0,C 180,E1 -5614.415,E2 -5614.415} C_VEL
LIN {X 0,Y 509.78,Z 122.6,A -85,B 0,C 180,E1 -5617.345,E2 -5617.345} C_VEL
LIN {X 0,Y 509.818,Z 122.599,A -85,B 0,C 180,E1 -5620.385,E2 -5620.385} C_VEL
LIN {X 0,Y 509.81,Z 122.6,A -85,B 0,C 180,E1 -5623.573,E2 -5623.573} C_VEL
LIN {X 0,Y 509.81,Z 122.598,A -85,B 0,C 180,E1 -5626.427,E2 -5626.427} C_VEL
LIN {X 0,Y 509.817,Z 122.601,A -85,B 0,C 180,E1 -5629.615,E2 -5629.615} C_VEL
LIN {X 0,Y 509.812,Z 122.604,A -85,B 0,C 180,E1 -5632.658,E2 -5632.658} C_VEL
LIN {X 0,Y 509.812,Z 122.6,A -85,B 0,C 180,E1 -5633.693,E2 -5633.693} C_VEL
LIN {X 0,Y 509.144,Z 122.691,A -85,B 0,C 180,E1 -5634.353,E2 -5634.353} C_VEL
LIN {X 0,Y 506.322,Z 123.038,A -85,B 0,C 180,E1 -5635.425,E2 -5635.425} C_VEL
LIN {X 0,Y 503.93,Z 123.341,A -85,B 0,C 180,E1 -5636.288,E2 -5636.288} C_VEL
LIN {X 0,Y 502.888,Z 123.462,A -85,B 0,C 180,E1 -5636.954,E2 -5636.954} C_VEL
LIN {X 0,Y 502.794,Z 123.472,A -85,B 0,C 180,E1 -5637.18,E2 -5637.18} C_VEL
LIN {X 0,Y 502.816,Z 123.479,A -85,B 0,C 180,E1 -5640.066,E2 -5640.066} C_VEL
LIN {X 0,Y 502.789,Z 123.478,A -85,B 0,C 180,E1 -5643.429,E2 -5643.429} C_VEL
LIN {X 0,Y 502.772,Z 123.487,A -85,B 0,C 180,E1 -5646.085,E2 -5646.085} C_VEL
LIN {X 0,Y 502.787,Z 123.478,A -85,B 0,C 180,E1 -5648.689,E2 -5648.689} C_VEL
LIN {X 0,Y 502.817,Z 123.472,A -85,B 0,C 180,E1 -5651.247,E2 -5651.247} C_VEL
LIN {X 0,Y 502.844,Z 123.471,A -85,B 0,C 180,E1 -5654.663,E2 -5654.663} C_VEL
LIN {X 0,Y 502.883,Z 123.471,A -85,B 0,C 180,E1 -5658.039,E2 -5658.039} C_VEL
LIN {X 0,Y 502.868,Z 123.472,A -85,B 0,C 180,E1 -5661.156,E2 -5661.156} C_VEL
LIN {X 0,Y 502.938,Z 123.644,A -85,B 0,C 180,E1 -5663.468,E2 -5663.468} C_VEL
LIN {X 0,Y 505.346,Z 134.886,A -85,B 0,C 180,E1 -5665.413,E2 -5665.413} C_VEL
LIN {X 0,Y 505.267,Z 142.798,A -85,B 0,C 180,E1 -5666.661,E2 -5666.661} C_VEL
LIN {X 0,Y 508.718,Z 157.8,A -85,B 0,C 180,E1 -5667.045,E2 -5667.045} C_VEL
LIN {X 0,Y 507.543,Z 306.67,A -85,B 0,C 180,E1 -5669.231,E2 -5669.231} C_VEL
LIN {X 0,Y 507.244,Z 321.925,A -85,B 0,C 180,E1 -5669.603,E2 -5669.603} C_VEL
LIN {X 0,Y 506.823,Z 336.166,A -85,B 0,C 180,E1 -5670.104,E2 -5670.104} C_VEL
LIN {X 0,Y 506.325,Z 349.732,A -85,B 0,C 180,E1 -5670.731,E2 -5670.731} C_VEL
LIN {X 0,Y 505.78,Z 362.875,A -85,B 0,C 180,E1 -5671.493,E2 -5671.493} C_VEL
LIN {X 0,Y 505.166,Z 375.589,A -85,B 0,C 180,E1 -5672.392,E2 -5672.392} C_VEL
LIN {X 0,Y 504.53,Z 388.412,A -85,B 0,C 180,E1 -5673.494,E2 -5673.494} C_VEL
LIN {X 0,Y 504.028,Z 399.165,A -85,B 0,C 180,E1 -5674.598,E2 -5674.598} C_VEL
LIN {X 0,Y 503.516,Z 409.164,A -85,B 0,C 180,E1 -5675.808,E2 -5675.808} C_VEL
LIN {X 0,Y 503.075,Z 419.446,A -85,B 0,C 180,E1 -5677.304,E2 -5677.304} C_VEL
LIN {X 0,Y 502.67,Z 428.181,A -85,B 0,C 180,E1 -5678.847,E2 -5678.847} C_VEL
LIN {X 0,Y 502.419,Z 435.677,A -85,B 0,C 180,E1 -5680.477,E2 -5680.477} C_VEL
LIN {X 0,Y 502.251,Z 441.666,A -85,B 0,C 180,E1 -5682.116,E2 -5682.116} C_VEL
LIN {X 0,Y 502.118,Z 446.279,A -85,B 0,C 180,E1 -5683.765,E2 -5683.765} C_VEL
LIN {X 0,Y 502.003,Z 449.591,A -85,B 0,C 180,E1 -5685.426,E2 -5685.426} C_VEL
LIN {X 0,Y 502.012,Z 451.628,A -85,B 0,C 180,E1 -5687.097,E2 -5687.097} C_VEL
LIN {X 0,Y 501.98,Z 452.439,A -85,B 0,C 180,E1 -5688.784,E2 -5688.784} C_VEL
LIN {X 0,Y 502.011,Z 451.997,A -85,B 0,C 180,E1 -5690.487,E2 -5690.487} C_VEL
LIN {X 0,Y 502.022,Z 450.257,A -85,B 0,C 180,E1 -5692.209,E2 -5692.209} C_VEL
LIN {X 0,Y 502.097,Z 447.133,A -85,B 0,C 180,E1 -5693.949,E2 -5693.949} C_VEL
LIN {X 0,Y 502.214,Z 443.853,A -85,B 0,C 180,E1 -5695.266,E2 -5695.266} C_VEL
LIN {X 0,Y 502.312,Z 439.576,A -85,B 0,C 180,E1 -5696.597,E2 -5696.597} C_VEL
LIN {X 0,Y 502.524,Z 433.08,A -85,B 0,C 180,E1 -5698.226,E2 -5698.226} C_VEL
LIN {X 0,Y 502.79,Z 426.251,A -85,B 0,C 180,E1 -5699.618,E2 -5699.618} C_VEL
LIN {X 0,Y 503.154,Z 417.368,A -85,B 0,C 180,E1 -5701.118,E2 -5701.118} C_VEL
LIN {X 0,Y 503.629,Z 407.54,A -85,B 0,C 180,E1 -5702.497,E2 -5702.497} C_VEL
LIN {X 0,Y 504.12,Z 397.446,A -85,B 0,C 180,E1 -5703.692,E2 -5703.692} C_VEL
LIN {X 0,Y 504.706,Z 386.198,A -85,B 0,C 180,E1 -5704.814,E2 -5704.814} C_VEL
LIN {X 0,Y 505.318,Z 372.953,A -85,B 0,C 180,E1 -5705.913,E2 -5705.913} C_VEL
LIN {X 0,Y 505.928,Z 359.871,A -85,B 0,C 180,E1 -5706.803,E2 -5706.803} C_VEL
LIN {X 0,Y 506.501,Z 345.954,A -85,B 0,C 180,E1 -5707.565,E2 -5707.565} C_VEL
LIN {X 0,Y 506.98,Z 331.49,A -85,B 0,C 180,E1 -5708.181,E2 -5708.181} C_VEL
LIN {X 0,Y 507.359,Z 316.273,A -85,B 0,C 180,E1 -5708.657,E2 -5708.657} C_VEL
LIN {X 0,Y 507.608,Z 300.634,A -85,B 0,C 180,E1 -5708.974,E2 -5708.974} C_VEL
LIN {X 0,Y 508.83,Z 158.075,A -85,B 0,C 180,E1 -5711.059,E2 -5711.059} C_VEL
LIN {X 0,Y 505.339,Z 142.763,A -85,B 0,C 180,E1 -5711.483,E2 -5711.483} C_VEL
LIN {X 0,Y 505.531,Z 136.164,A -85,B 0,C 180,E1 -5712.538,E2 -5712.538} C_VEL
LIN {X 0,Y 502.824,Z 123.478,A -85,B 0,C 180,E1 -5714.787,E2 -5714.787} C_VEL
LIN {X 0,Y 502.797,Z 123.483,A -85,B 0,C 180,E1 -5717.86,E2 -5717.86} C_VEL
LIN {X 0,Y 502.8,Z 123.481,A -85,B 0,C 180,E1 -5721.023,E2 -5721.023} C_VEL
LIN {X 0,Y 502.773,Z 123.486,A -85,B 0,C 180,E1 -5724.169,E2 -5724.169} C_VEL
LIN {X 0,Y 502.834,Z 123.472,A -85,B 0,C 180,E1 -5726.993,E2 -5726.993} C_VEL
LIN {X 0,Y 502.815,Z 123.481,A -85,B 0,C 180,E1 -5730.065,E2 -5730.065} C_VEL
LIN {X 0,Y 502.845,Z 123.471,A -85,B 0,C 180,E1 -5733.443,E2 -5733.443} C_VEL
LIN {X 0,Y 502.788,Z 123.474,A -85,B 0,C 180,E1 -5736.959,E2 -5736.959} C_VEL
LIN {X 0,Y 502.837,Z 123.474,A -85,B 0,C 180,E1 -5739.548,E2 -5739.548} C_VEL
LIN {X 0,Y 502.818,Z 123.477,A -85,B 0,C 180,E1 -5742.091,E2 -5742.091} C_VEL
LIN {X 0,Y 502.834,Z 123.473,A -85,B 0,C 180,E1 -5745.428,E2 -5745.428} C_VEL
LIN {X 0,Y 502.878,Z 123.464,A -85,B 0,C 180,E1 -5748.716,E2 -5748.716} C_VEL
LIN {X 0,Y 502.901,Z 123.466,A -85,B 0,C 180,E1 -5751.966,E2 -5751.966} C_VEL
LIN {X 0,Y 502.932,Z 123.456,A -85,B 0,C 180,E1 -5754.386,E2 -5754.386} C_VEL
LIN {X 0,Y 503.026,Z 123.45,A -85,B 0,C 180,E1 -5757.597,E2 -5757.597} C_VEL
LIN {X 0,Y 503.028,Z 123.448,A -85,B 0,C 180,E1 -5760,E2 -5760} C_VEL
LIN {X 0,Y 503.024,Z 123.446,A -85,B 0,C 180,E1 -5762.402,E2 -5762.402} C_VEL
LIN {X 0,Y 502.93,Z 123.462,A -85,B 0,C 180,E1 -5765.613,E2 -5765.613} C_VEL
LIN {X 0,Y 502.864,Z 123.47,A -85,B 0,C 180,E1 -5768.843,E2 -5768.843} C_VEL
LIN {X 0,Y 502.846,Z 123.467,A -85,B 0,C 180,E1 -5772.101,E2 -5772.101} C_VEL
LIN {X 0,Y 502.848,Z 123.469,A -85,B 0,C 180,E1 -5775.399,E2 -5775.399} C_VEL
LIN {X 0,Y 502.825,Z 123.478,A -85,B 0,C 180,E1 -5778.752,E2 -5778.752} C_VEL
LIN {X 0,Y 502.783,Z 123.48,A -85,B 0,C 180,E1 -5781.311,E2 -5781.311} C_VEL
LIN {X 0,Y 502.784,Z 123.476,A -85,B 0,C 180,E1 -5783.914,E2 -5783.914} C_VEL
LIN {X 0,Y 502.863,Z 123.471,A -85,B 0,C 180,E1 -5786.566,E2 -5786.566} C_VEL
LIN {X 0,Y 502.822,Z 123.472,A -85,B 0,C 180,E1 -5789.288,E2 -5789.288} C_VEL
LIN {X 0,Y 502.781,Z 123.479,A -85,B 0,C 180,E1 -5792.085,E2 -5792.085} C_VEL
LIN {X 0,Y 502.794,Z 123.478,A -85,B 0,C 180,E1 -5794.966,E2 -5794.966} C_VEL
LIN {X 0,Y 502.792,Z 123.477,A -85,B 0,C 180,E1 -5797.954,E2 -5797.954} C_VEL
LIN {X 0,Y 502.818,Z 123.475,A -85,B 0,C 180,E1 -5801.066,E2 -5801.066} C_VEL
LIN {X 0,Y 502.8,Z 123.481,A -85,B 0,C 180,E1 -5804.532,E2 -5804.532} C_VEL
LIN {X 0,Y 502.794,Z 123.478,A -85,B 0,C 180,E1 -5807.861,E2 -5807.861} C_VEL
LIN {X 0,Y 502.801,Z 123.477,A -85,B 0,C 180,E1 -5811.024,E2 -5811.024} C_VEL
LIN {X 0,Y 502.773,Z 123.484,A -85,B 0,C 180,E1 -5814.169,E2 -5814.169} C_VEL
LIN {X 0,Y 502.831,Z 123.471,A -85,B 0,C 180,E1 -5816.993,E2 -5816.993} C_VEL
LIN {X 0,Y 502.814,Z 123.479,A -85,B 0,C 180,E1 -5820.065,E2 -5820.065} C_VEL
LIN {X 0,Y 502.88,Z 123.653,A -85,B 0,C 180,E1 -5821.146,E2 -5821.146} C_VEL
LIN {X 0,Y 506.241,Z 138.108,A -85,B 0,C 180,E1 -5823.439,E2 -5823.439} C_VEL
LIN {X 0,Y 505.813,Z 151.897,A -85,B 0,C 180,E1 -5825.365,E2 -5825.365} C_VEL
LIN {X 0,Y 505.16,Z 167.911,A -85,B 0,C 180,E1 -5827.56,E2 -5827.56} C_VEL
LIN {X 0,Y 508.721,Z 186.875,A -85,B 0,C 180,E1 -5828.021,E2 -5828.021} C_VEL
LIN {X 0,Y 507.43,Z 333.644,A -85,B 0,C 180,E1 -5830.177,E2 -5830.177} C_VEL
LIN {X 0,Y 507.018,Z 349.641,A -85,B 0,C 180,E1 -5830.569,E2 -5830.569} C_VEL
LIN {X 0,Y 506.557,Z 364.476,A -85,B 0,C 180,E1 -5831.102,E2 -5831.102} C_VEL
LIN {X 0,Y 505.962,Z 378.947,A -85,B 0,C 180,E1 -5831.788,E2 -5831.788} C_VEL
LIN {X 0,Y 505.373,Z 392.516,A -85,B 0,C 180,E1 -5832.603,E2 -5832.603} C_VEL
LIN {X 0,Y 504.749,Z 406.32,A -85,B 0,C 180,E1 -5833.623,E2 -5833.623} C_VEL
LIN {X 0,Y 504.131,Z 418.817,A -85,B 0,C 180,E1 -5834.744,E2 -5834.744} C_VEL
LIN {X 0,Y 503.632,Z 429.305,A -85,B 0,C 180,E1 -5835.865,E2 -5835.865} C_VEL
LIN {X 0,Y 503.177,Z 439.038,A -85,B 0,C 180,E1 -5837.087,E2 -5837.087} C_VEL
LIN {X 0,Y 502.781,Z 448.804,A -85,B 0,C 180,E1 -5838.545,E2 -5838.545} C_VEL
LIN {X 0,Y 502.52,Z 456.558,A -85,B 0,C 180,E1 -5839.932,E2 -5839.932} C_VEL
LIN {X 0,Y 502.318,Z 463.992,A -85,B 0,C 180,E1 -5841.553,E2 -5841.553} C_VEL
LIN {X 0,Y 502.201,Z 469.89,A -85,B 0,C 180,E1 -5843.169,E2 -5843.169} C_VEL
LIN {X 0,Y 502.175,Z 473.394,A -85,B 0,C 180,E1 -5844.378,E2 -5844.378} C_VEL
LIN {X 0,Y 502.069,Z 476.935,A -85,B 0,C 180,E1 -5845.987,E2 -5845.987} C_VEL
LIN {X 0,Y 502.088,Z 479.267,A -85,B 0,C 180,E1 -5847.594,E2 -5847.594} C_VEL
LIN {X 0,Y 501.987,Z 480.439,A -85,B 0,C 180,E1 -5849.198,E2 -5849.198} C_VEL
LIN {X 0,Y 501.987,Z 480.442,A -85,B 0,C 180,E1 -5850.803,E2 -5850.803} C_VEL
LIN {X 0,Y 502.088,Z 479.273,A -85,B 0,C 180,E1 -5852.407,E2 -5852.407} C_VEL
LIN {X 0,Y 502.069,Z 476.946,A -85,B 0,C 180,E1 -5854.014,E2 -5854.014} C_VEL
LIN {X 0,Y 502.176,Z 473.418,A -85,B 0,C 180,E1 -5855.622,E2 -5855.622} C_VEL
LIN {X 0,Y 502.238,Z 468.593,A -85,B 0,C 180,E1 -5857.235,E2 -5857.235} C_VEL
LIN {X 0,Y 502.363,Z 462.342,A -85,B 0,C 180,E1 -5858.853,E2 -5858.853} C_VEL
LIN {X 0,Y 502.636,Z 454.493,A -85,B 0,C 180,E1 -5860.473,E2 -5860.473} C_VEL
LIN {X 0,Y 502.901,Z 445.622,A -85,B 0,C 180,E1 -5861.974,E2 -5861.974} C_VEL
LIN {X 0,Y 503.342,Z 436.082,A -85,B 0,C 180,E1 -5863.32,E2 -5863.32} C_VEL
LIN {X 0,Y 503.798,Z 425.798,A -85,B 0,C 180,E1 -5864.543,E2 -5864.543} C_VEL
LIN {X 0,Y 504.396,Z 413.737,A -85,B 0,C 180,E1 -5865.747,E2 -5865.747} C_VEL
LIN {X 0,Y 505,Z 401.231,A -85,B 0,C 180,E1 -5866.785,E2 -5866.785} C_VEL
LIN {X 0,Y 505.657,Z 387.829,A -85,B 0,C 180,E1 -5867.701,E2 -5867.701} C_VEL
LIN {X 0,Y 506.17,Z 375.007,A -85,B 0,C 180,E1 -5868.414,E2 -5868.414} C_VEL
LIN {X 0,Y 506.699,Z 360.657,A -85,B 0,C 180,E1 -5869.048,E2 -5869.048} C_VEL
LIN {X 0,Y 507.085,Z 345.97,A -85,B 0,C 180,E1 -5869.533,E2 -5869.533} C_VEL
LIN {X 0,Y 507.44,Z 330.069,A -85,B 0,C 180,E1 -5869.881,E2 -5869.881} C_VEL
LIN {X 0,Y 508.672,Z 186.817,A -85,B 0,C 180,E1 -5871.967,E2 -5871.967} C_VEL
LIN {X 0,Y 505.135,Z 168.067,A -85,B 0,C 180,E1 -5872.423,E2 -5872.423} C_VEL
LIN {X 0,Y 505.997,Z 147.683,A -85,B 0,C 180,E1 -5875.201,E2 -5875.201} C_VEL
LIN {X 0,Y 506.215,Z 137.89,A -85,B 0,C 180,E1 -5876.561,E2 -5876.561} C_VEL
LIN {X 0,Y 502.829,Z 123.476,A -85,B 0,C 180,E1 -5878.829,E2 -5878.829} C_VEL
LIN {X 0,Y 502.785,Z 123.485,A -85,B 0,C 180,E1 -5882.085,E2 -5882.085} C_VEL
LIN {X 0,Y 502.801,Z 123.479,A -85,B 0,C 180,E1 -5884.966,E2 -5884.966} C_VEL
LIN {X 0,Y 502.795,Z 123.481,A -85,B 0,C 180,E1 -5887.954,E2 -5887.954} C_VEL
LIN {X 0,Y 502.802,Z 123.477,A -85,B 0,C 180,E1 -5891.068,E2 -5891.068} C_VEL
LIN {X 0,Y 502.781,Z 123.48,A -85,B 0,C 180,E1 -5894.341,E2 -5894.341} C_VEL
LIN {X 0,Y 502.774,Z 123.48,A -85,B 0,C 180,E1 -5896.769,E2 -5896.769} C_VEL
LIN {X 0,Y 502.821,Z 123.476,A -85,B 0,C 180,E1 -5899.006,E2 -5899.006} C_VEL
LIN {X 0,Y 502.795,Z 123.476,A -85,B 0,C 180,E1 -5902.046,E2 -5902.046} C_VEL
LIN {X 0,Y 502.798,Z 123.479,A -85,B 0,C 180,E1 -5905.034,E2 -5905.034} C_VEL
LIN {X 0,Y 502.785,Z 123.477,A -85,B 0,C 180,E1 -5907.916,E2 -5907.916} C_VEL
LIN {X 0,Y 502.808,Z 123.476,A -85,B 0,C 180,E1 -5910.711,E2 -5910.711} C_VEL
LIN {X 0,Y 502.847,Z 123.468,A -85,B 0,C 180,E1 -5913.444,E2 -5913.444} C_VEL
LIN {X 0,Y 502.79,Z 123.482,A -85,B 0,C 180,E1 -5916.96,E2 -5916.96} C_VEL
LIN {X 0,Y 502.838,Z 123.47,A -85,B 0,C 180,E1 -5919.549,E2 -5919.549} C_VEL
LIN {X 0,Y 502.821,Z 123.472,A -85,B 0,C 180,E1 -5922.092,E2 -5922.092} C_VEL
LIN {X 0,Y 502.83,Z 123.472,A -85,B 0,C 180,E1 -5925.429,E2 -5925.429} C_VEL
LIN {X 0,Y 502.88,Z 123.471,A -85,B 0,C 180,E1 -5928.717,E2 -5928.717} C_VEL
LIN {X 0,Y 502.861,Z 123.468,A -85,B 0,C 180,E1 -5931.966,E2 -5931.966} C_VEL
LIN {X 0,Y 502.897,Z 123.471,A -85,B 0,C 180,E1 -5934.386,E2 -5934.386} C_VEL
LIN {X 0,Y 503.013,Z 123.445,A -85,B 0,C 180,E1 -5937.598,E2 -5937.598} C_VEL
LIN {X 0,Y 503.007,Z 123.442,A -85,B 0,C 180,E1 -5940,E2 -5940} C_VEL
LIN {X 0,Y 503.012,Z 123.451,A -85,B 0,C 180,E1 -5942.403,E2 -5942.403} C_VEL
LIN {X 0,Y 502.895,Z 123.465,A -85,B 0,C 180,E1 -5945.614,E2 -5945.614} C_VEL
LIN {X 0,Y 502.851,Z 123.465,A -85,B 0,C 180,E1 -5948.034,E2 -5948.034} C_VEL
LIN {X 0,Y 502.84,Z 123.464,A -85,B 0,C 180,E1 -5951.284,E2 -5951.284} C_VEL
LIN {X 0,Y 502.802,Z 123.474,A -85,B 0,C 180,E1 -5954.572,E2 -5954.572} C_VEL
LIN {X 0,Y 502.775,Z 123.482,A -85,B 0,C 180,E1 -5957.911,E2 -5957.911} C_VEL
LIN {X 0,Y 502.773,Z 123.477,A -85,B 0,C 180,E1 -5960.517,E2 -5960.517} C_VEL
LIN {X 0,Y 502.761,Z 123.48,A -85,B 0,C 180,E1 -5963.043,E2 -5963.043} C_VEL
LIN {X 0,Y 502.762,Z 123.482,A -85,B 0,C 180,E1 -5965.68,E2 -5965.68} C_VEL
LIN {X 0,Y 502.764,Z 123.472,A -85,B 0,C 180,E1 -5968.378,E2 -5968.378} C_VEL
LIN {X 0,Y 502.77,Z 123.481,A -85,B 0,C 180,E1 -5971.493,E2 -5971.493} C_VEL
LIN {X 0,Y 502.784,Z 123.477,A -85,B 0,C 180,E1 -5974.44,E2 -5974.44} C_VEL
LIN {X 0,Y 502.734,Z 123.48,A -85,B 0,C 180,E1 -5977.17,E2 -5977.17} C_VEL
LIN {X 0,Y 502.773,Z 123.474,A -85,B 0,C 180,E1 -5980.017,E2 -5980.017} C_VEL
LIN {X 0,Y 502.751,Z 123.482,A -85,B 0,C 180,E1 -5983.234,E2 -5983.234} C_VEL
LIN {X 0,Y 502.783,Z 123.469,A -85,B 0,C 180,E1 -5985.66,E2 -5985.66} C_VEL
LIN {X 0,Y 502.768,Z 123.483,A -85,B 0,C 180,E1 -5989.013,E2 -5989.013} C_VEL
LIN {X 0,Y 502.777,Z 123.476,A -85,B 0,C 180,E1 -5992.044,E2 -5992.044} C_VEL
LIN {X 0,Y 502.797,Z 123.477,A -85,B 0,C 180,E1 -5995.033,E2 -5995.033} C_VEL
LIN {X 0,Y 502.794,Z 123.472,A -85,B 0,C 180,E1 -5997.18,E2 -5997.18} C_VEL
LIN {X 0,Y 502.107,Z 123.56,A -85,B 0,C 180,E1 -5997.849,E2 -5997.849} C_VEL
LIN {X 0,Y 499.255,Z 123.919,A -85,B 0,C 180,E1 -5998.935,E2 -5998.935} C_VEL
LIN {X 0,Y 496.854,Z 124.222,A -85,B 0,C 180,E1 -5999.81,E2 -5999.81} C_VEL
LIN {X 0,Y 495.819,Z 124.35,A -85,B 0,C 180,E1 -6000.486,E2 -6000.486} C_VEL
LIN {X 0,Y 495.732,Z 124.357,A -85,B 0,C 180,E1 -6000.714,E2 -6000.714} C_VEL
LIN {X 0,Y 495.723,Z 124.363,A -85,B 0,C 180,E1 -6003.928,E2 -6003.928} C_VEL
LIN {X 0,Y 495.764,Z 124.353,A -85,B 0,C 180,E1 -6007.14,E2 -6007.14} C_VEL
LIN {X 0,Y 495.773,Z 124.356,A -85,B 0,C 180,E1 -6010.109,E2 -6010.109} C_VEL
LIN {X 0,Y 495.75,Z 124.35,A -85,B 0,C 180,E1 -6012.68,E2 -6012.68} C_VEL
LIN {X 0,Y 495.787,Z 124.351,A -85,B 0,C 180,E1 -6015.217,E2 -6015.217} C_VEL
LIN {X 0,Y 495.857,Z 124.343,A -85,B 0,C 180,E1 -6018.555,E2 -6018.555} C_VEL
LIN {X 0,Y 495.836,Z 124.349,A -85,B 0,C 180,E1 -6021.851,E2 -6021.851} C_VEL
LIN {X 0,Y 495.872,Z 124.421,A -85,B 0,C 180,E1 -6023.193,E2 -6023.193} C_VEL
LIN {X 0,Y 498.514,Z 136.712,A -85,B 0,C 180,E1 -6025.35,E2 -6025.35} C_VEL
LIN {X 0,Y 498.48,Z 143.149,A -85,B 0,C 180,E1 -6026.349,E2 -6026.349} C_VEL
LIN {X 0,Y 502.182,Z 159.141,A -85,B 0,C 180,E1 -6026.765,E2 -6026.765} C_VEL
LIN {X 0,Y 500.848,Z 307.342,A -85,B 0,C 180,E1 -6028.97,E2 -6028.97} C_VEL
LIN {X 0,Y 500.475,Z 323.317,A -85,B 0,C 180,E1 -6029.371,E2 -6029.371} C_VEL
LIN {X 0,Y 500.012,Z 338.889,A -85,B 0,C 180,E1 -6029.949,E2 -6029.949} C_VEL
LIN {X 0,Y 499.441,Z 353.306,A -85,B 0,C 180,E1 -6030.66,E2 -6030.66} C_VEL
LIN {X 0,Y 498.785,Z 367.051,A -85,B 0,C 180,E1 -6031.513,E2 -6031.513} C_VEL
LIN {X 0,Y 498.135,Z 380.282,A -85,B 0,C 180,E1 -6032.527,E2 -6032.527} C_VEL
LIN {X 0,Y 497.474,Z 392.365,A -85,B 0,C 180,E1 -6033.645,E2 -6033.645} C_VEL
LIN {X 0,Y 496.892,Z 403.407,A -85,B 0,C 180,E1 -6034.868,E2 -6034.868} C_VEL
LIN {X 0,Y 496.335,Z 414.211,A -85,B 0,C 180,E1 -6036.3,E2 -6036.3} C_VEL
LIN {X 0,Y 495.936,Z 422.955,A -85,B 0,C 180,E1 -6037.696,E2 -6037.696} C_VEL
LIN {X 0,Y 495.596,Z 429.7,A -85,B 0,C 180,E1 -6038.974,E2 -6038.974} C_VEL
LIN {X 0,Y 495.336,Z 436.941,A -85,B 0,C 180,E1 -6040.629,E2 -6040.629} C_VEL
LIN {X 0,Y 495.145,Z 442.691,A -85,B 0,C 180,E1 -6042.293,E2 -6042.293} C_VEL
LIN {X 0,Y 495.036,Z 447.073,A -85,B 0,C 180,E1 -6043.966,E2 -6043.966} C_VEL
LIN {X 0,Y 494.9,Z 450.183,A -85,B 0,C 180,E1 -6045.653,E2 -6045.653} C_VEL
LIN {X 0,Y 494.904,Z 452.049,A -85,B 0,C 180,E1 -6047.35,E2 -6047.35} C_VEL
LIN {X 0,Y 494.889,Z 452.684,A -85,B 0,C 180,E1 -6049.064,E2 -6049.064} C_VEL
LIN {X 0,Y 494.909,Z 452.031,A -85,B 0,C 180,E1 -6050.794,E2 -6050.794} C_VEL
LIN {X 0,Y 494.947,Z 449.937,A -85,B 0,C 180,E1 -6052.635,E2 -6052.635} C_VEL
LIN {X 0,Y 495.047,Z 446.697,A -85,B 0,C 180,E1 -6054.312,E2 -6054.312} C_VEL
LIN {X 0,Y 495.2,Z 441.811,A -85,B 0,C 180,E1 -6056.101,E2 -6056.101} C_VEL
LIN {X 0,Y 495.336,Z 436.998,A -85,B 0,C 180,E1 -6057.459,E2 -6057.459} C_VEL
LIN {X 0,Y 495.604,Z 430.05,A -85,B 0,C 180,E1 -6059.057,E2 -6059.057} C_VEL
LIN {X 0,Y 496.01,Z 421.399,A -85,B 0,C 180,E1 -6060.669,E2 -6060.669} C_VEL
LIN {X 0,Y 496.482,Z 411.793,A -85,B 0,C 180,E1 -6062.142,E2 -6062.142} C_VEL
LIN {X 0,Y 497.037,Z 401.437,A -85,B 0,C 180,E1 -6063.466,E2 -6063.466} C_VEL
LIN {X 0,Y 497.551,Z 390.891,A -85,B 0,C 180,E1 -6064.606,E2 -6064.606} C_VEL
LIN {X 0,Y 498.221,Z 378.744,A -85,B 0,C 180,E1 -6065.707,E2 -6065.707} C_VEL
LIN {X 0,Y 498.862,Z 366.069,A -85,B 0,C 180,E1 -6066.662,E2 -6066.662} C_VEL
LIN {X 0,Y 499.518,Z 352.733,A -85,B 0,C 180,E1 -6067.482,E2 -6067.482} C_VEL
LIN {X 0,Y 500.041,Z 337.987,A -85,B 0,C 180,E1 -6068.2,E2 -6068.2} C_VEL
LIN {X 0,Y 500.531,Z 322.36,A -85,B 0,C 180,E1 -6068.766,E2 -6068.766} C_VEL
LIN {X 0,Y 500.898,Z 307.534,A -85,B 0,C 180,E1 -6069.136,E2 -6069.136} C_VEL
LIN {X 0,Y 502.291,Z 159.404,A -85,B 0,C 180,E1 -6071.351,E2 -6071.351} C_VEL
LIN {X 0,Y 498.561,Z 142.995,A -85,B 0,C 180,E1 -6071.813,E2 -6071.813} C_VEL
LIN {X 0,Y 498.729,Z 138.357,A -85,B 0,C 180,E1 -6072.563,E2 -6072.563} C_VEL
LIN {X 0,Y 496.645,Z 128.148,A -85,B 0,C 180,E1 -6074.387,E2 -6074.387} C_VEL
LIN {X 0,Y 495.773,Z 124.355,A -85,B 0,C 180,E1 -6075.086,E2 -6075.086} C_VEL
LIN {X 0,Y 495.751,Z 124.36,A -85,B 0,C 180,E1 -6078.218,E2 -6078.218} C_VEL
LIN {X 0,Y 495.75,Z 124.359,A -85,B 0,C 180,E1 -6081.408,E2 -6081.408} C_VEL
LIN {X 0,Y 495.747,Z 124.356,A -85,B 0,C 180,E1 -6084.462,E2 -6084.462} C_VEL
LIN {X 0,Y 495.769,Z 124.352,A -85,B 0,C 180,E1 -6087.405,E2 -6087.405} C_VEL
LIN {X 0,Y 495.764,Z 124.356,A -85,B 0,C 180,E1 -6090.253,E2 -6090.253} C_VEL
LIN {X 0,Y 495.776,Z 124.351,A -85,B 0,C 180,E1 -6093.262,E2 -6093.262} C_VEL
LIN {X 0,Y 495.741,Z 124.353,A -85,B 0,C 180,E1 -6096.612,E2 -6096.612} C_VEL
LIN {X 0,Y 495.78,Z 124.351,A -85,B 0,C 180,E1 -6099.324,E2 -6099.324} C_VEL
LIN {X 0,Y 495.78,Z 124.355,A -85,B 0,C 180,E1 -6101.828,E2 -6101.828} C_VEL
LIN {X 0,Y 495.824,Z 124.343,A -85,B 0,C 180,E1 -6104.548,E2 -6104.548} C_VEL
LIN {X 0,Y 495.829,Z 124.347,A -85,B 0,C 180,E1 -6107.965,E2 -6107.965} C_VEL
LIN {X 0,Y 495.838,Z 124.343,A -85,B 0,C 180,E1 -6111.03,E2 -6111.03} C_VEL
LIN {X 0,Y 495.861,Z 124.346,A -85,B 0,C 180,E1 -6113.489,E2 -6113.489} C_VEL
LIN {X 0,Y 495.838,Z 124.343,A -85,B 0,C 180,E1 -6116.749,E2 -6116.749} C_VEL
LIN {X 0,Y 495.867,Z 124.336,A -85,B 0,C 180,E1 -6118.375,E2 -6118.375} C_VEL
LIN {X 0,Y 495.983,Z 124.326,A -85,B 0,C 180,E1 -6120.812,E2 -6120.812} C_VEL
LIN {X 0,Y 495.993,Z 124.322,A -85,B 0,C 180,E1 -6122.436,E2 -6122.436} C_VEL
LIN {X 0,Y 495.885,Z 124.338,A -85,B 0,C 180,E1 -6125.693,E2 -6125.693} C_VEL
LIN {X 0,Y 495.834,Z 124.346,A -85,B 0,C 180,E1 -6128.97,E2 -6128.97} C_VEL
LIN {X 0,Y 495.828,Z 124.342,A -85,B 0,C 180,E1 -6132.035,E2 -6132.035} C_VEL
LIN {X 0,Y 495.823,Z 124.344,A -85,B 0,C 180,E1 -6135.451,E2 -6135.451} C_VEL
LIN {X 0,Y 495.778,Z 124.351,A -85,B 0,C 180,E1 -6138.237,E2 -6138.237} C_VEL
LIN {X 0,Y 495.774,Z 124.355,A -85,B 0,C 180,E1 -6140.756,E2 -6140.756} C_VEL
LIN {X 0,Y 495.747,Z 124.355,A -85,B 0,C 180,E1 -6143.387,E2 -6143.387} C_VEL
LIN {X 0,Y 495.79,Z 124.348,A -85,B 0,C 180,E1 -6146.068,E2 -6146.068} C_VEL
LIN {X 0,Y 495.77,Z 124.354,A -85,B 0,C 180,E1 -6148.815,E2 -6148.815} C_VEL
LIN {X 0,Y 495.754,Z 124.353,A -85,B 0,C 180,E1 -6151.725,E2 -6151.725} C_VEL
LIN {X 0,Y 495.761,Z 124.356,A -85,B 0,C 180,E1 -6154.693,E2 -6154.693} C_VEL
LIN {X 0,Y 495.728,Z 124.355,A -85,B 0,C 180,E1 -6157.562,E2 -6157.562} C_VEL
LIN {X 0,Y 495.765,Z 124.357,A -85,B 0,C 180,E1 -6160.7,E2 -6160.7} C_VEL
LIN {X 0,Y 495.733,Z 124.355,A -85,B 0,C 180,E1 -6164.001,E2 -6164.001} C_VEL
LIN {X 0,Y 495.724,Z 124.354,A -85,B 0,C 180,E1 -6167.117,E2 -6167.117} C_VEL
LIN {X 0,Y 495.758,Z 124.355,A -85,B 0,C 180,E1 -6169.953,E2 -6169.953} C_VEL
LIN {X 0,Y 495.727,Z 124.358,A -85,B 0,C 180,E1 -6172.553,E2 -6172.553} C_VEL
LIN {X 0,Y 495.776,Z 124.351,A -85,B 0,C 180,E1 -6175.457,E2 -6175.457} C_VEL
LIN {X 0,Y 495.754,Z 124.356,A -85,B 0,C 180,E1 -6178.364,E2 -6178.364} C_VEL
LIN {X 0,Y 495.811,Z 124.428,A -85,B 0,C 180,E1 -6180.811,E2 -6180.811} C_VEL
LIN {X 0,Y 499.316,Z 139.357,A -85,B 0,C 180,E1 -6183.23,E2 -6183.23} C_VEL
LIN {X 0,Y 499.492,Z 142.467,A -85,B 0,C 180,E1 -6183.691,E2 -6183.691} C_VEL
LIN {X 0,Y 498.508,Z 164.26,A -85,B 0,C 180,E1 -6186.75,E2 -6186.75} C_VEL
LIN {X 0,Y 498.332,Z 167.647,A -85,B 0,C 180,E1 -6187.218,E2 -6187.218} C_VEL
LIN {X 0,Y 502.161,Z 187.356,A -85,B 0,C 180,E1 -6187.723,E2 -6187.723} C_VEL
LIN {X 0,Y 500.737,Z 334.3,A -85,B 0,C 180,E1 -6189.916,E2 -6189.916} C_VEL
LIN {X 0,Y 500.299,Z 350.107,A -85,B 0,C 180,E1 -6190.318,E2 -6190.318} C_VEL
LIN {X 0,Y 499.811,Z 364.753,A -85,B 0,C 180,E1 -6190.856,E2 -6190.856} C_VEL
LIN {X 0,Y 499.206,Z 378.768,A -85,B 0,C 180,E1 -6191.533,E2 -6191.533} C_VEL
LIN {X 0,Y 498.572,Z 392.331,A -85,B 0,C 180,E1 -6192.358,E2 -6192.358} C_VEL
LIN {X 0,Y 497.945,Z 404.835,A -85,B 0,C 180,E1 -6193.288,E2 -6193.288} C_VEL
LIN {X 0,Y 497.27,Z 417.548,A -85,B 0,C 180,E1 -6194.423,E2 -6194.423} C_VEL
LIN {X 0,Y 496.668,Z 429.099,A -85,B 0,C 180,E1 -6195.663,E2 -6195.663} C_VEL
LIN {X 0,Y 496.171,Z 438.824,A -85,B 0,C 180,E1 -6196.901,E2 -6196.901} C_VEL
LIN {X 0,Y 495.771,Z 448.34,A -85,B 0,C 180,E1 -6198.34,E2 -6198.34} C_VEL
LIN {X 0,Y 495.487,Z 456.345,A -85,B 0,C 180,E1 -6199.788,E2 -6199.788} C_VEL
LIN {X 0,Y 495.23,Z 463.781,A -85,B 0,C 180,E1 -6201.431,E2 -6201.431} C_VEL
LIN {X 0,Y 495.116,Z 469.682,A -85,B 0,C 180,E1 -6203.07,E2 -6203.07} C_VEL
LIN {X 0,Y 495.07,Z 473.188,A -85,B 0,C 180,E1 -6204.297,E2 -6204.297} C_VEL
LIN {X 0,Y 494.967,Z 476.732,A -85,B 0,C 180,E1 -6205.929,E2 -6205.929} C_VEL
LIN {X 0,Y 494.993,Z 479.067,A -85,B 0,C 180,E1 -6207.559,E2 -6207.559} C_VEL
LIN {X 0,Y 494.907,Z 480.241,A -85,B 0,C 180,E1 -6209.187,E2 -6209.187} C_VEL
LIN {X 0,Y 494.907,Z 480.244,A -85,B 0,C 180,E1 -6210.814,E2 -6210.814} C_VEL
LIN {X 0,Y 494.994,Z 479.075,A -85,B 0,C 180,E1 -6212.442,E2 -6212.442} C_VEL
LIN {X 0,Y 494.967,Z 476.747,A -85,B 0,C 180,E1 -6214.071,E2 -6214.071} C_VEL
LIN {X 0,Y 495.073,Z 473.218,A -85,B 0,C 180,E1 -6215.703,E2 -6215.703} C_VEL
LIN {X 0,Y 495.157,Z 468.392,A -85,B 0,C 180,E1 -6217.339,E2 -6217.339} C_VEL
LIN {X 0,Y 495.287,Z 462.139,A -85,B 0,C 180,E1 -6218.98,E2 -6218.98} C_VEL
LIN {X 0,Y 495.598,Z 454.288,A -85,B 0,C 180,E1 -6220.624,E2 -6220.624} C_VEL
LIN {X 0,Y 495.872,Z 445.991,A -85,B 0,C 180,E1 -6222.058,E2 -6222.058} C_VEL
LIN {X 0,Y 496.378,Z 435.871,A -85,B 0,C 180,E1 -6223.51,E2 -6223.51} C_VEL
LIN {X 0,Y 496.849,Z 425.575,A -85,B 0,C 180,E1 -6224.751,E2 -6224.751} C_VEL
LIN {X 0,Y 497.529,Z 413.121,A -85,B 0,C 180,E1 -6226.006,E2 -6226.006} C_VEL
LIN {X 0,Y 498.167,Z 399.601,A -85,B 0,C 180,E1 -6227.128,E2 -6227.128} C_VEL
LIN {X 0,Y 498.881,Z 385.871,A -85,B 0,C 180,E1 -6228.055,E2 -6228.055} C_VEL
LIN {X 0,Y 499.556,Z 371.628,A -85,B 0,C 180,E1 -6228.826,E2 -6228.826} C_VEL
LIN {X 0,Y 500.078,Z 356.508,A -85,B 0,C 180,E1 -6229.46,E2 -6229.46} C_VEL
LIN {X 0,Y 500.514,Z 341.444,A -85,B 0,C 180,E1 -6229.916,E2 -6229.916} C_VEL
LIN {X 0,Y 500.803,Z 325.964,A -85,B 0,C 180,E1 -6230.217,E2 -6230.217} C_VEL
LIN {X 0,Y 502.069,Z 187.318,A -85,B 0,C 180,E1 -6232.256,E2 -6232.256} C_VEL
LIN {X 0,Y 498.29,Z 167.829,A -85,B 0,C 180,E1 -6232.748,E2 -6232.748} C_VEL
LIN {X 0,Y 499.161,Z 148.95,A -85,B 0,C 180,E1 -6235.352,E2 -6235.352} C_VEL
LIN {X 0,Y 499.47,Z 140.511,A -85,B 0,C 180,E1 -6236.536,E2 -6236.536} C_VEL
LIN {X 0,Y 496.457,Z 127.067,A -85,B 0,C 180,E1 -6238.635,E2 -6238.635} C_VEL
LIN {X 0,Y 495.791,Z 124.353,A -85,B 0,C 180,E1 -6239.104,E2 -6239.104} C_VEL
LIN {X 0,Y 495.769,Z 124.357,A -85,B 0,C 180,E1 -6242.595,E2 -6242.595} C_VEL
LIN {X 0,Y 495.75,Z 124.361,A -85,B 0,C 180,E1 -6245.538,E2 -6245.538} C_VEL
LIN {X 0,Y 495.766,Z 124.352,A -85,B 0,C 180,E1 -6248.769,E2 -6248.769} C_VEL
LIN {X 0,Y 495.752,Z 124.361,A -85,B 0,C 180,E1 -6251.782,E2 -6251.782} C_VEL
LIN {X 0,Y 495.74,Z 124.359,A -85,B 0,C 180,E1 -6255.141,E2 -6255.141} C_VEL
LIN {X 0,Y 495.758,Z 124.354,A -85,B 0,C 180,E1 -6258.219,E2 -6258.219} C_VEL
LIN {X 0,Y 495.75,Z 124.357,A -85,B 0,C 180,E1 -6261.409,E2 -6261.409} C_VEL
LIN {X 0,Y 495.75,Z 124.352,A -85,B 0,C 180,E1 -6264.463,E2 -6264.463} C_VEL
LIN {X 0,Y 495.769,Z 124.356,A -85,B 0,C 180,E1 -6267.406,E2 -6267.406} C_VEL
LIN {X 0,Y 495.76,Z 124.35,A -85,B 0,C 180,E1 -6270.254,E2 -6270.254} C_VEL
LIN {X 0,Y 495.777,Z 124.35,A -85,B 0,C 180,E1 -6273.263,E2 -6273.263} C_VEL
LIN {X 0,Y 495.742,Z 124.357,A -85,B 0,C 180,E1 -6276.613,E2 -6276.613} C_VEL
LIN {X 0,Y 495.783,Z 124.351,A -85,B 0,C 180,E1 -6279.325,E2 -6279.325} C_VEL
LIN {X 0,Y 495.783,Z 124.348,A -85,B 0,C 180,E1 -6281.829,E2 -6281.829} C_VEL
LIN {X 0,Y 495.781,Z 124.351,A -85,B 0,C 180,E1 -6285.217,E2 -6285.217} C_VEL
LIN {X 0,Y 495.855,Z 124.345,A -85,B 0,C 180,E1 -6288.555,E2 -6288.555} C_VEL
LIN {X 0,Y 495.824,Z 124.344,A -85,B 0,C 180,E1 -6291.852,E2 -6291.852} C_VEL
LIN {X 0,Y 495.856,Z 124.346,A -85,B 0,C 180,E1 -6294.306,E2 -6294.306} C_VEL
LIN {X 0,Y 495.98,Z 124.321,A -85,B 0,C 180,E1 -6297.564,E2 -6297.564} C_VEL
LIN {X 0,Y 495.976,Z 124.317,A -85,B 0,C 180,E1 -6300,E2 -6300} C_VEL
LIN {X 0,Y 495.979,Z 124.327,A -85,B 0,C 180,E1 -6302.437,E2 -6302.437} C_VEL
LIN {X 0,Y 495.854,Z 124.343,A -85,B 0,C 180,E1 -6305.694,E2 -6305.694} C_VEL
LIN {X 0,Y 495.815,Z 124.339,A -85,B 0,C 180,E1 -6308.149,E2 -6308.149} C_VEL
LIN {X 0,Y 495.818,Z 124.339,A -85,B 0,C 180,E1 -6311.446,E2 -6311.446} C_VEL
LIN {X 0,Y 495.75,Z 124.353,A -85,B 0,C 180,E1 -6314.784,E2 -6314.784} C_VEL
LIN {X 0,Y 495.739,Z 124.355,A -85,B 0,C 180,E1 -6318.174,E2 -6318.174} C_VEL
LIN {X 0,Y 495.723,Z 124.36,A -85,B 0,C 180,E1 -6321.63,E2 -6321.63} C_VEL
LIN {X 0,Y 495.697,Z 124.36,A -85,B 0,C 180,E1 -6324.278,E2 -6324.278} C_VEL
LIN {X 0,Y 495.722,Z 124.358,A -85,B 0,C 180,E1 -6326.98,E2 -6326.98} C_VEL
LIN {X 0,Y 495.7,Z 124.352,A -85,B 0,C 180,E1 -6329.751,E2 -6329.751} C_VEL
LIN {X 0,Y 495.729,Z 124.355,A -85,B 0,C 180,E1 -6332.598,E2 -6332.598} C_VEL
LIN {X 0,Y 495.724,Z 124.356,A -85,B 0,C 180,E1 -6335.54,E2 -6335.54} C_VEL
LIN {X 0,Y 495.739,Z 124.349,A -85,B 0,C 180,E1 -6338.764,E2 -6338.764} C_VEL
LIN {X 0,Y 495.728,Z 124.356,A -85,B 0,C 180,E1 -6341.785,E2 -6341.785} C_VEL
LIN {X 0,Y 495.743,Z 124.349,A -85,B 0,C 180,E1 -6345.141,E2 -6345.141} C_VEL
LIN {X 0,Y 495.728,Z 124.357,A -85,B 0,C 180,E1 -6348.215,E2 -6348.215} C_VEL
LIN {X 0,Y 495.748,Z 124.351,A -85,B 0,C 180,E1 -6351.235,E2 -6351.235} C_VEL
LIN {X 0,Y 495.748,Z 124.36,A -85,B 0,C 180,E1 -6354.462,E2 -6354.462} C_VEL
LIN {X 0,Y 495.757,Z 124.348,A -85,B 0,C 180,E1 -6357.404,E2 -6357.404} C_VEL
LIN {X 0,Y 495.763,Z 124.36,A -85,B 0,C 180,E1 -6360.253,E2 -6360.253} C_VEL
LIN {X 0,Y 495.732,Z 124.357,A -85,B 0,C 180,E1 -6360.714,E2 -6360.714} C_VEL
LIN {X 0,Y 495.05,Z 124.441,A -85,B 0,C 180,E1 -6361.393,E2 -6361.393} C_VEL
LIN {X 0,Y 492.174,Z 124.805,A -85,B 0,C 180,E1 -6362.495,E2 -6362.495} C_VEL
LIN {X 0,Y 489.766,Z 125.102,A -85,B 0,C 180,E1 -6363.383,E2 -6363.383} C_VEL
LIN {X 0,Y 488.756,Z 125.233,A -85,B 0,C 180,E1 -6364.069,E2 -6364.069} C_VEL
LIN {X 0,Y 488.687,Z 125.238,A -85,B 0,C 180,E1 -6364.301,E2 -6364.301} C_VEL
LIN {X 0,Y 488.726,Z 125.23,A -85,B 0,C 180,E1 -6367.153,E2 -6367.153} C_VEL
LIN {X 0,Y 488.729,Z 125.234,A -85,B 0,C 180,E1 -6369.81,E2 -6369.81} C_VEL
LIN {X 0,Y 488.707,Z 125.228,A -85,B 0,C 180,E1 -6372.422,E2 -6372.422} C_VEL
LIN {X 0,Y 488.762,Z 125.225,A -85,B 0,C 180,E1 -6374.999,E2 -6374.999} C_VEL
LIN {X 0,Y 488.811,Z 125.222,A -85,B 0,C 180,E1 -6378.387,E2 -6378.387} C_VEL
LIN {X 0,Y 488.785,Z 125.228,A -85,B 0,C 180,E1 -6381.733,E2 -6381.733} C_VEL
LIN {X 0,Y 488.813,Z 125.224,A -85,B 0,C 180,E1 -6382.914,E2 -6382.914} C_VEL
LIN {X 0,Y 491.205,Z 136.164,A -85,B 0,C 180,E1 -6384.869,E2 -6384.869} C_VEL
LIN {X 0,Y 491.732,Z 139.773,A -85,B 0,C 180,E1 -6385.491,E2 -6385.491} C_VEL
LIN {X 0,Y 491.616,Z 142.996,A -85,B 0,C 180,E1 -6386.013,E2 -6386.013} C_VEL
LIN {X 0,Y 495.597,Z 160.364,A -85,B 0,C 180,E1 -6386.481,E2 -6386.481} C_VEL
LIN {X 0,Y 494.168,Z 307.855,A -85,B 0,C 180,E1 -6388.701,E2 -6388.701} C_VEL
LIN {X 0,Y 493.766,Z 323.725,A -85,B 0,C 180,E1 -6389.108,E2 -6389.108} C_VEL
LIN {X 0,Y 493.277,Z 339.255,A -85,B 0,C 180,E1 -6389.694,E2 -6389.694} C_VEL
LIN {X 0,Y 492.751,Z 352.206,A -85,B 0,C 180,E1 -6390.334,E2 -6390.334} C_VEL
LIN {X 0,Y 492.069,Z 365.924,A -85,B 0,C 180,E1 -6391.181,E2 -6391.181} C_VEL
LIN {X 0,Y 491.367,Z 378.729,A -85,B 0,C 180,E1 -6392.151,E2 -6392.151} C_VEL
LIN {X 0,Y 490.689,Z 391.082,A -85,B 0,C 180,E1 -6393.284,E2 -6393.284} C_VEL
LIN {X 0,Y 489.998,Z 402.38,A -85,B 0,C 180,E1 -6394.524,E2 -6394.524} C_VEL
LIN {X 0,Y 489.454,Z 411.925,A -85,B 0,C 180,E1 -6395.768,E2 -6395.768} C_VEL
LIN {X 0,Y 489.032,Z 420.924,A -85,B 0,C 180,E1 -6397.157,E2 -6397.157} C_VEL
LIN {X 0,Y 488.596,Z 429.196,A -85,B 0,C 180,E1 -6398.686,E2 -6398.686} C_VEL
LIN {X 0,Y 488.303,Z 436.575,A -85,B 0,C 180,E1 -6400.364,E2 -6400.364} C_VEL
LIN {X 0,Y 488.095,Z 442.453,A -85,B 0,C 180,E1 -6402.05,E2 -6402.05} C_VEL
LIN {X 0,Y 487.995,Z 445.954,A -85,B 0,C 180,E1 -6403.322,E2 -6403.322} C_VEL
LIN {X 0,Y 487.888,Z 449.723,A -85,B 0,C 180,E1 -6405.173,E2 -6405.173} C_VEL
LIN {X 0,Y 487.788,Z 451.742,A -85,B 0,C 180,E1 -6406.747,E2 -6406.747} C_VEL
LIN {X 0,Y 487.806,Z 452.778,A -85,B 0,C 180,E1 -6408.479,E2 -6408.479} C_VEL
LIN {X 0,Y 487.828,Z 452.567,A -85,B 0,C 180,E1 -6410.228,E2 -6410.228} C_VEL
LIN {X 0,Y 487.824,Z 451.064,A -85,B 0,C 180,E1 -6411.998,E2 -6411.998} C_VEL
LIN {X 0,Y 487.92,Z 448.19,A -85,B 0,C 180,E1 -6413.785,E2 -6413.785} C_VEL
LIN {X 0,Y 488.086,Z 443.827,A -85,B 0,C 180,E1 -6415.593,E2 -6415.593} C_VEL
LIN {X 0,Y 488.223,Z 439.101,A -85,B 0,C 180,E1 -6417.077,E2 -6417.077} C_VEL
LIN {X 0,Y 488.49,Z 432.844,A -85,B 0,C 180,E1 -6418.642,E2 -6418.642} C_VEL
LIN {X 0,Y 488.847,Z 425.15,A -85,B 0,C 180,E1 -6420.211,E2 -6420.211} C_VEL
LIN {X 0,Y 489.247,Z 416.802,A -85,B 0,C 180,E1 -6421.622,E2 -6421.622} C_VEL
LIN {X 0,Y 489.81,Z 406.776,A -85,B 0,C 180,E1 -6423.041,E2 -6423.041} C_VEL
LIN {X 0,Y 490.431,Z 395.697,A -85,B 0,C 180,E1 -6424.35,E2 -6424.35} C_VEL
LIN {X 0,Y 491.16,Z 383.303,A -85,B 0,C 180,E1 -6425.569,E2 -6425.569} C_VEL
LIN {X 0,Y 491.84,Z 370.346,A -85,B 0,C 180,E1 -6426.625,E2 -6426.625} C_VEL
LIN {X 0,Y 492.606,Z 356.226,A -85,B 0,C 180,E1 -6427.557,E2 -6427.557} C_VEL
LIN {X 0,Y 493.236,Z 342.077,A -85,B 0,C 180,E1 -6428.3,E2 -6428.3} C_VEL
LIN {X 0,Y 493.765,Z 326.963,A -85,B 0,C 180,E1 -6428.906,E2 -6428.906} C_VEL
LIN {X 0,Y 494.167,Z 311.484,A -85,B 0,C 180,E1 -6429.345,E2 -6429.345} C_VEL
LIN {X 0,Y 494.455,Z 290.99,A -85,B 0,C 180,E1 -6429.697,E2 -6429.697} C_VEL
LIN {X 0,Y 495.697,Z 160.328,A -85,B 0,C 180,E1 -6431.668,E2 -6431.668} C_VEL
LIN {X 0,Y 491.801,Z 143.265,A -85,B 0,C 180,E1 -6432.154,E2 -6432.154} C_VEL
LIN {X 0,Y 491.76,Z 138.844,A -85,B 0,C 180,E1 -6432.893,E2 -6432.893} C_VEL
LIN {X 0,Y 488.894,Z 126.172,A -85,B 0,C 180,E1 -6435.219,E2 -6435.219} C_VEL
LIN {X 0,Y 488.715,Z 125.234,A -85,B 0,C 180,E1 -6435.412,E2 -6435.412} C_VEL
LIN {X 0,Y 488.694,Z 125.241,A -85,B 0,C 180,E1 -6438.582,E2 -6438.582} C_VEL
LIN {X 0,Y 488.703,Z 125.239,A -85,B 0,C 180,E1 -6440.947,E2 -6440.947} C_VEL
LIN {X 0,Y 488.671,Z 125.241,A -85,B 0,C 180,E1 -6443.867,E2 -6443.867} C_VEL
LIN {X 0,Y 488.74,Z 125.228,A -85,B 0,C 180,E1 -6446.877,E2 -6446.877} C_VEL
LIN {X 0,Y 488.724,Z 125.233,A -85,B 0,C 180,E1 -6449.78,E2 -6449.78} C_VEL
LIN {X 0,Y 488.726,Z 125.229,A -85,B 0,C 180,E1 -6453.072,E2 -6453.072} C_VEL
LIN {X 0,Y 488.672,Z 125.233,A -85,B 0,C 180,E1 -6456.253,E2 -6456.253} C_VEL
LIN {X 0,Y 488.748,Z 125.227,A -85,B 0,C 180,E1 -6459.175,E2 -6459.175} C_VEL
LIN {X 0,Y 488.748,Z 125.232,A -85,B 0,C 180,E1 -6461.632,E2 -6461.632} C_VEL
LIN {X 0,Y 488.758,Z 125.223,A -85,B 0,C 180,E1 -6464.999,E2 -6464.999} C_VEL
LIN {X 0,Y 488.806,Z 125.218,A -85,B 0,C 180,E1 -6468.387,E2 -6468.387} C_VEL
LIN {X 0,Y 488.817,Z 125.222,A -85,B 0,C 180,E1 -6471.733,E2 -6471.733} C_VEL
LIN {X 0,Y 488.847,Z 125.211,A -85,B 0,C 180,E1 -6474.224,E2 -6474.224} C_VEL
LIN {X 0,Y 488.961,Z 125.202,A -85,B 0,C 180,E1 -6477.528,E2 -6477.528} C_VEL
LIN {X 0,Y 488.934,Z 125.204,A -85,B 0,C 180,E1 -6480.823,E2 -6480.823} C_VEL
LIN {X 0,Y 488.961,Z 125.198,A -85,B 0,C 180,E1 -6482.471,E2 -6482.471} C_VEL
LIN {X 0,Y 488.842,Z 125.215,A -85,B 0,C 180,E1 -6485.776,E2 -6485.776} C_VEL
LIN {X 0,Y 488.785,Z 125.22,A -85,B 0,C 180,E1 -6488.267,E2 -6488.267} C_VEL
LIN {X 0,Y 488.806,Z 125.218,A -85,B 0,C 180,E1 -6491.612,E2 -6491.612} C_VEL
LIN {X 0,Y 488.762,Z 125.23,A -85,B 0,C 180,E1 -6495,E2 -6495} C_VEL
LIN {X 0,Y 488.746,Z 125.228,A -85,B 0,C 180,E1 -6498.442,E2 -6498.442} C_VEL
LIN {X 0,Y 488.706,Z 125.236,A -85,B 0,C 180,E1 -6501.07,E2 -6501.07} C_VEL
LIN {X 0,Y 488.688,Z 125.232,A -85,B 0,C 180,E1 -6503.745,E2 -6503.745} C_VEL
LIN {X 0,Y 488.791,Z 125.226,A -85,B 0,C 180,E1 -6506.943,E2 -6506.943} C_VEL
LIN {X 0,Y 488.708,Z 125.234,A -85,B 0,C 180,E1 -6510.363,E2 -6510.363} C_VEL
LIN {X 0,Y 488.728,Z 125.229,A -85,B 0,C 180,E1 -6513.483,E2 -6513.483} C_VEL
LIN {X 0,Y 488.681,Z 125.241,A -85,B 0,C 180,E1 -6516.354,E2 -6516.354} C_VEL
LIN {X 0,Y 488.699,Z 125.228,A -85,B 0,C 180,E1 -6519.254,E2 -6519.254} C_VEL
LIN {X 0,Y 488.705,Z 125.233,A -85,B 0,C 180,E1 -6521.6,E2 -6521.6} C_VEL
LIN {X 0,Y 488.711,Z 125.233,A -85,B 0,C 180,E1 -6524.801,E2 -6524.801} C_VEL
LIN {X 0,Y 488.69,Z 125.231,A -85,B 0,C 180,E1 -6527.475,E2 -6527.475} C_VEL
LIN {X 0,Y 488.731,Z 125.23,A -85,B 0,C 180,E1 -6529.677,E2 -6529.677} C_VEL
LIN {X 0,Y 488.678,Z 125.235,A -85,B 0,C 180,E1 -6532.841,E2 -6532.841} C_VEL
LIN {X 0,Y 488.729,Z 125.233,A -85,B 0,C 180,E1 -6535.887,E2 -6535.887} C_VEL
LIN {X 0,Y 488.691,Z 125.235,A -85,B 0,C 180,E1 -6538.82,E2 -6538.82} C_VEL
LIN {X 0,Y 488.751,Z 125.412,A -85,B 0,C 180,E1 -6540.495,E2 -6540.495} C_VEL
LIN {X 0,Y 492.158,Z 139.303,A -85,B 0,C 180,E1 -6542.809,E2 -6542.809} C_VEL
LIN {X 0,Y 492.697,Z 143.968,A -85,B 0,C 180,E1 -6543.528,E2 -6543.528} C_VEL
LIN {X 0,Y 491.596,Z 166.146,A -85,B 0,C 180,E1 -6546.687,E2 -6546.687} C_VEL
LIN {X 0,Y 491.525,Z 167.492,A -85,B 0,C 180,E1 -6546.876,E2 -6546.876} C_VEL
LIN {X 0,Y 495.548,Z 188.088,A -85,B 0,C 180,E1 -6547.412,E2 -6547.412} C_VEL
LIN {X 0,Y 494.113,Z 333.801,A -85,B 0,C 180,E1 -6549.62,E2 -6549.62} C_VEL
LIN {X 0,Y 493.645,Z 349.519,A -85,B 0,C 180,E1 -6550.021,E2 -6550.021} C_VEL
LIN {X 0,Y 493.087,Z 365.036,A -85,B 0,C 180,E1 -6550.601,E2 -6550.601} C_VEL
LIN {X 0,Y 492.447,Z 378.643,A -85,B 0,C 180,E1 -6551.27,E2 -6551.27} C_VEL
LIN {X 0,Y 491.783,Z 392.16,A -85,B 0,C 180,E1 -6552.106,E2 -6552.106} C_VEL
LIN {X 0,Y 491.064,Z 404.645,A -85,B 0,C 180,E1 -6553.046,E2 -6553.046} C_VEL
LIN {X 0,Y 490.358,Z 417.356,A -85,B 0,C 180,E1 -6554.198,E2 -6554.198} C_VEL
LIN {X 0,Y 489.7,Z 428.906,A -85,B 0,C 180,E1 -6555.454,E2 -6555.454} C_VEL
LIN {X 0,Y 489.185,Z 438.63,A -85,B 0,C 180,E1 -6556.711,E2 -6556.711} C_VEL
LIN {X 0,Y 488.743,Z 448.412,A -85,B 0,C 180,E1 -6558.215,E2 -6558.215} C_VEL
LIN {X 0,Y 488.456,Z 456.144,A -85,B 0,C 180,E1 -6559.639,E2 -6559.639} C_VEL
LIN {X 0,Y 488.151,Z 463.576,A -85,B 0,C 180,E1 -6561.306,E2 -6561.306} C_VEL
LIN {X 0,Y 488.046,Z 469.476,A -85,B 0,C 180,E1 -6562.97,E2 -6562.97} C_VEL
LIN {X 0,Y 487.97,Z 472.983,A -85,B 0,C 180,E1 -6564.214,E2 -6564.214} C_VEL
LIN {X 0,Y 487.868,Z 476.529,A -85,B 0,C 180,E1 -6565.87,E2 -6565.87} C_VEL
LIN {X 0,Y 487.903,Z 478.866,A -85,B 0,C 180,E1 -6567.524,E2 -6567.524} C_VEL
LIN {X 0,Y 487.83,Z 480.042,A -85,B 0,C 180,E1 -6569.175,E2 -6569.175} C_VEL
LIN {X 0,Y 487.83,Z 480.046,A -85,B 0,C 180,E1 -6570.826,E2 -6570.826} C_VEL
LIN {X 0,Y 487.904,Z 478.877,A -85,B 0,C 180,E1 -6572.477,E2 -6572.477} C_VEL
LIN {X 0,Y 487.868,Z 476.549,A -85,B 0,C 180,E1 -6574.131,E2 -6574.131} C_VEL
LIN {X 0,Y 487.975,Z 473.018,A -85,B 0,C 180,E1 -6575.787,E2 -6575.787} C_VEL
LIN {X 0,Y 488.06,Z 468.19,A -85,B 0,C 180,E1 -6577.447,E2 -6577.447} C_VEL
LIN {X 0,Y 488.222,Z 461.933,A -85,B 0,C 180,E1 -6579.111,E2 -6579.111} C_VEL
LIN {X 0,Y 488.572,Z 454.074,A -85,B 0,C 180,E1 -6580.778,E2 -6580.778} C_VEL
LIN {X 0,Y 488.842,Z 445.912,A -85,B 0,C 180,E1 -6582.211,E2 -6582.211} C_VEL
LIN {X 0,Y 489.405,Z 435.629,A -85,B 0,C 180,E1 -6583.707,E2 -6583.707} C_VEL
LIN {X 0,Y 489.91,Z 425.328,A -85,B 0,C 180,E1 -6584.965,E2 -6584.965} C_VEL
LIN {X 0,Y 490.597,Z 413.67,A -85,B 0,C 180,E1 -6586.159,E2 -6586.159} C_VEL
LIN {X 0,Y 491.248,Z 400.697,A -85,B 0,C 180,E1 -6587.269,E2 -6587.269} C_VEL
LIN {X 0,Y 492.014,Z 387.254,A -85,B 0,C 180,E1 -6588.208,E2 -6588.208} C_VEL
LIN {X 0,Y 492.645,Z 374.389,A -85,B 0,C 180,E1 -6588.939,E2 -6588.939} C_VEL
LIN {X 0,Y 493.23,Z 360.188,A -85,B 0,C 180,E1 -6589.58,E2 -6589.58} C_VEL
LIN {X 0,Y 493.707,Z 345.489,A -85,B 0,C 180,E1 -6590.075,E2 -6590.075} C_VEL
LIN {X 0,Y 494.084,Z 330.081,A -85,B 0,C 180,E1 -6590.423,E2 -6590.423} C_VEL
LIN {X 0,Y 495.474,Z 188.152,A -85,B 0,C 180,E1 -6592.545,E2 -6592.545} C_VEL
LIN {X 0,Y 491.478,Z 167.741,A -85,B 0,C 180,E1 -6593.056,E2 -6593.056} C_VEL
LIN {X 0,Y 492.422,Z 147.096,A -85,B 0,C 180,E1 -6595.953,E2 -6595.953} C_VEL
LIN {X 0,Y 492.561,Z 141.799,A -85,B 0,C 180,E1 -6596.709,E2 -6596.709} C_VEL
LIN {X 0,Y 488.747,Z 125.232,A -85,B 0,C 180,E1 -6599.358,E2 -6599.358} C_VEL
LIN {X 0,Y 488.705,Z 125.238,A -85,B 0,C 180,E1 -6602.147,E2 -6602.147} C_VEL
LIN {X 0,Y 488.719,Z 125.234,A -85,B 0,C 180,E1 -6605.115,E2 -6605.115} C_VEL
LIN {X 0,Y 488.682,Z 125.238,A -85,B 0,C 180,E1 -6608.2,E2 -6608.2} C_VEL
LIN {X 0,Y 488.72,Z 125.232,A -85,B 0,C 180,E1 -6610.345,E2 -6610.345} C_VEL
LIN {X 0,Y 488.68,Z 125.243,A -85,B 0,C 180,E1 -6613.656,E2 -6613.656} C_VEL
LIN {X 0,Y 488.686,Z 125.236,A -85,B 0,C 180,E1 -6616.346,E2 -6616.346} C_VEL
LIN {X 0,Y 488.736,Z 125.231,A -85,B 0,C 180,E1 -6619.677,E2 -6619.677} C_VEL
LIN {X 0,Y 488.681,Z 125.235,A -85,B 0,C 180,E1 -6622.842,E2 -6622.842} C_VEL
LIN {X 0,Y 488.727,Z 125.229,A -85,B 0,C 180,E1 -6625.887,E2 -6625.887} C_VEL
LIN {X 0,Y 488.692,Z 125.235,A -85,B 0,C 180,E1 -6628.821,E2 -6628.821} C_VEL
LIN {X 0,Y 488.701,Z 125.223,A -85,B 0,C 180,E1 -6631.669,E2 -6631.669} C_VEL
LIN {X 0,Y 488.709,Z 125.227,A -85,B 0,C 180,E1 -6634.442,E2 -6634.442} C_VEL
LIN {X 0,Y 488.724,Z 125.231,A -85,B 0,C 180,E1 -6637.154,E2 -6637.154} C_VEL
LIN {X 0,Y 488.727,Z 125.227,A -85,B 0,C 180,E1 -6639.811,E2 -6639.811} C_VEL
LIN {X 0,Y 488.711,Z 125.233,A -85,B 0,C 180,E1 -6642.423,E2 -6642.423} C_VEL
LIN {X 0,Y 488.758,Z 125.228,A -85,B 0,C 180,E1 -6645,E2 -6645} C_VEL
LIN {X 0,Y 488.81,Z 125.221,A -85,B 0,C 180,E1 -6648.388,E2 -6648.388} C_VEL
LIN {X 0,Y 488.775,Z 125.221,A -85,B 0,C 180,E1 -6651.733,E2 -6651.733} C_VEL
LIN {X 0,Y 488.816,Z 125.222,A -85,B 0,C 180,E1 -6654.224,E2 -6654.224} C_VEL
LIN {X 0,Y 488.946,Z 125.197,A -85,B 0,C 180,E1 -6657.529,E2 -6657.529} C_VEL
LIN {X 0,Y 488.945,Z 125.192,A -85,B 0,C 180,E1 -6660,E2 -6660} C_VEL
LIN {X 0,Y 488.945,Z 125.203,A -85,B 0,C 180,E1 -6662.472,E2 -6662.472} C_VEL
LIN {X 0,Y 488.814,Z 125.221,A -85,B 0,C 180,E1 -6665.777,E2 -6665.777} C_VEL
LIN {X 0,Y 488.759,Z 125.215,A -85,B 0,C 180,E1 -6668.268,E2 -6668.268} C_VEL
LIN {X 0,Y 488.779,Z 125.218,A -85,B 0,C 180,E1 -6671.613,E2 -6671.613} C_VEL
LIN {X 0,Y 488.719,Z 125.229,A -85,B 0,C 180,E1 -6675.002,E2 -6675.002} C_VEL
LIN {X 0,Y 488.681,Z 125.233,A -85,B 0,C 180,E1 -6678.445,E2 -6678.445} C_VEL
LIN {X 0,Y 488.68,Z 125.235,A -85,B 0,C 180,E1 -6681.072,E2 -6681.072} C_VEL
LIN {X 0,Y 488.653,Z 125.242,A -85,B 0,C 180,E1 -6683.748,E2 -6683.748} C_VEL
LIN {X 0,Y 488.672,Z 125.233,A -85,B 0,C 180,E1 -6686.477,E2 -6686.477} C_VEL
LIN {X 0,Y 488.664,Z 125.229,A -85,B 0,C 180,E1 -6689.275,E2 -6689.275} C_VEL
LIN {X 0,Y 488.683,Z 125.231,A -85,B 0,C 180,E1 -6692.149,E2 -6692.149} C_VEL
LIN {X 0,Y 488.705,Z 125.236,A -85,B 0,C 180,E1 -6695.117,E2 -6695.117} C_VEL
LIN {X 0,Y 488.656,Z 125.226,A -85,B 0,C 180,E1 -6698.203,E2 -6698.203} C_VEL
LIN {X 0,Y 488.699,Z 125.229,A -85,B 0,C 180,E1 -6700.341,E2 -6700.341} C_VEL
LIN {X 0,Y 488.678,Z 125.232,A -85,B 0,C 180,E1 -6703.656,E2 -6703.656} C_VEL
LIN {X 0,Y 488.678,Z 125.228,A -85,B 0,C 180,E1 -6706.344,E2 -6706.344} C_VEL
LIN {X 0,Y 488.709,Z 125.23,A -85,B 0,C 180,E1 -6709.674,E2 -6709.674} C_VEL
LIN {X 0,Y 488.672,Z 125.237,A -85,B 0,C 180,E1 -6712.84,E2 -6712.84} C_VEL
LIN {X 0,Y 488.723,Z 125.23,A -85,B 0,C 180,E1 -6715.886,E2 -6715.886} C_VEL
LIN {X 0,Y 488.695,Z 125.236,A -85,B 0,C 180,E1 -6718.82,E2 -6718.82} C_VEL
LIN {X 0,Y 488.7,Z 125.232,A -85,B 0,C 180,E1 -6721.668,E2 -6721.668} C_VEL
LIN {X 0,Y 488.687,Z 125.238,A -85,B 0,C 180,E1 -6724.301,E2 -6724.301} C_VEL
LIN {X 0,Y 488.054,Z 125.322,A -85,B 0,C 180,E1 -6724.989,E2 -6724.989} C_VEL
LIN {X 0,Y 485.213,Z 125.678,A -85,B 0,C 180,E1 -6726.106,E2 -6726.106} C_VEL
LIN {X 0,Y 482.783,Z 125.977,A -85,B 0,C 180,E1 -6727.007,E2 -6727.007} C_VEL
LIN {X 0,Y 481.731,Z 126.104,A -85,B 0,C 180,E1 -6727.702,E2 -6727.702} C_VEL
LIN {X 0,Y 481.641,Z 126.114,A -85,B 0,C 180,E1 -6727.938,E2 -6727.938} C_VEL
LIN {X 0,Y 481.706,Z 126.105,A -85,B 0,C 180,E1 -6730.393,E2 -6730.393} C_VEL
LIN {X 0,Y 481.673,Z 126.103,A -85,B 0,C 180,E1 -6733.033,E2 -6733.033} C_VEL
LIN {X 0,Y 481.688,Z 126.107,A -85,B 0,C 180,E1 -6735.638,E2 -6735.638} C_VEL
LIN {X 0,Y 481.757,Z 126.101,A -85,B 0,C 180,E1 -6738.215,E2 -6738.215} C_VEL
LIN {X 0,Y 481.741,Z 126.107,A -85,B 0,C 180,E1 -6741.611,E2 -6741.611} C_VEL
LIN {X 0,Y 481.805,Z 126.192,A -85,B 0,C 180,E1 -6742.666,E2 -6742.666} C_VEL
LIN {X 0,Y 484.397,Z 137.985,A -85,B 0,C 180,E1 -6744.797,E2 -6744.797} C_VEL
LIN {X 0,Y 484.881,Z 141.609,A -85,B 0,C 180,E1 -6745.427,E2 -6745.427} C_VEL
LIN {X 0,Y 484.836,Z 143.407,A -85,B 0,C 180,E1 -6745.7,E2 -6745.7} C_VEL
LIN {X 0,Y 489.005,Z 162.162,A -85,B 0,C 180,E1 -6746.198,E2 -6746.198} C_VEL
LIN {X 0,Y 487.492,Z 308.102,A -85,B 0,C 180,E1 -6748.425,E2 -6748.425} C_VEL
LIN {X 0,Y 487.06,Z 323.961,A -85,B 0,C 180,E1 -6748.837,E2 -6748.837} C_VEL
LIN {X 0,Y 486.545,Z 339.479,A -85,B 0,C 180,E1 -6749.431,E2 -6749.431} C_VEL
LIN {X 0,Y 485.977,Z 352.743,A -85,B 0,C 180,E1 -6750.096,E2 -6750.096} C_VEL
LIN {X 0,Y 485.286,Z 366.099,A -85,B 0,C 180,E1 -6750.933,E2 -6750.933} C_VEL
LIN {X 0,Y 484.506,Z 379.624,A -85,B 0,C 180,E1 -6751.974,E2 -6751.974} C_VEL
LIN {X 0,Y 483.767,Z 391.889,A -85,B 0,C 180,E1 -6753.123,E2 -6753.123} C_VEL
LIN {X 0,Y 483.062,Z 403.094,A -85,B 0,C 180,E1 -6754.38,E2 -6754.38} C_VEL
LIN {X 0,Y 482.492,Z 412.553,A -85,B 0,C 180,E1 -6755.642,E2 -6755.642} C_VEL
LIN {X 0,Y 481.976,Z 422.248,A -85,B 0,C 180,E1 -6757.183,E2 -6757.183} C_VEL
LIN {X 0,Y 481.575,Z 429.688,A -85,B 0,C 180,E1 -6758.603,E2 -6758.603} C_VEL
LIN {X 0,Y 481.258,Z 436.206,A -85,B 0,C 180,E1 -6760.092,E2 -6760.092} C_VEL
LIN {X 0,Y 481.05,Z 442.208,A -85,B 0,C 180,E1 -6761.802,E2 -6761.802} C_VEL
LIN {X 0,Y 480.882,Z 446.835,A -85,B 0,C 180,E1 -6763.523,E2 -6763.523} C_VEL
LIN {X 0,Y 480.793,Z 450.152,A -85,B 0,C 180,E1 -6765.255,E2 -6765.255} C_VEL
LIN {X 0,Y 480.695,Z 452.21,A -85,B 0,C 180,E1 -6767.002,E2 -6767.002} C_VEL
LIN {X 0,Y 480.711,Z 453.032,A -85,B 0,C 180,E1 -6768.762,E2 -6768.762} C_VEL
LIN {X 0,Y 480.748,Z 452.529,A -85,B 0,C 180,E1 -6770.672,E2 -6770.672} C_VEL
LIN {X 0,Y 480.755,Z 450.874,A -85,B 0,C 180,E1 -6772.339,E2 -6772.339} C_VEL
LIN {X 0,Y 480.855,Z 447.761,A -85,B 0,C 180,E1 -6774.157,E2 -6774.157} C_VEL
LIN {X 0,Y 481.058,Z 443.145,A -85,B 0,C 180,E1 -6775.994,E2 -6775.994} C_VEL
LIN {X 0,Y 481.183,Z 438.618,A -85,B 0,C 180,E1 -6777.391,E2 -6777.391} C_VEL
LIN {X 0,Y 481.453,Z 432.765,A -85,B 0,C 180,E1 -6778.853,E2 -6778.853} C_VEL
LIN {X 0,Y 481.848,Z 425.167,A -85,B 0,C 180,E1 -6780.413,E2 -6780.413} C_VEL
LIN {X 0,Y 482.32,Z 416.67,A -85,B 0,C 180,E1 -6781.863,E2 -6781.863} C_VEL
LIN {X 0,Y 482.949,Z 406.435,A -85,B 0,C 180,E1 -6783.322,E2 -6783.322} C_VEL
LIN {X 0,Y 483.619,Z 395.266,A -85,B 0,C 180,E1 -6784.65,E2 -6784.65} C_VEL
LIN {X 0,Y 484.387,Z 383.294,A -85,B 0,C 180,E1 -6785.836,E2 -6785.836} C_VEL
LIN {X 0,Y 485.108,Z 370.183,A -85,B 0,C 180,E1 -6786.915,E2 -6786.915} C_VEL
LIN {X 0,Y 485.87,Z 356.921,A -85,B 0,C 180,E1 -6787.802,E2 -6787.802} C_VEL
LIN {X 0,Y 486.566,Z 342.108,A -85,B 0,C 180,E1 -6788.593,E2 -6788.593} C_VEL
LIN {X 0,Y 487.122,Z 326.994,A -85,B 0,C 180,E1 -6789.205,E2 -6789.205} C_VEL
LIN {X 0,Y 487.555,Z 311.617,A -85,B 0,C 180,E1 -6789.644,E2 -6789.644} C_VEL
LIN {X 0,Y 487.852,Z 290.41,A -85,B 0,C 180,E1 -6790.012,E2 -6790.012} C_VEL
LIN {X 0,Y 489.288,Z 161.89,A -85,B 0,C 180,E1 -6791.977,E2 -6791.977} C_VEL
LIN {X 0,Y 485.039,Z 143.441,A -85,B 0,C 180,E1 -6792.522,E2 -6792.522} C_VEL
LIN {X 0,Y 484.845,Z 140.178,A -85,B 0,C 180,E1 -6793.085,E2 -6793.085} C_VEL
LIN {X 0,Y 482.167,Z 128.287,A -85,B 0,C 180,E1 -6795.308,E2 -6795.308} C_VEL
LIN {X 0,Y 481.652,Z 126.116,A -85,B 0,C 180,E1 -6795.756,E2 -6795.756} C_VEL
LIN {X 0,Y 481.649,Z 126.119,A -85,B 0,C 180,E1 -6798.957,E2 -6798.957} C_VEL
LIN {X 0,Y 481.651,Z 126.117,A -85,B 0,C 180,E1 -6801.993,E2 -6801.993} C_VEL
LIN {X 0,Y 481.689,Z 126.102,A -85,B 0,C 180,E1 -6805.317,E2 -6805.317} C_VEL
LIN {X 0,Y 481.646,Z 126.111,A -85,B 0,C 180,E1 -6808.311,E2 -6808.311} C_VEL
LIN {X 0,Y 481.676,Z 126.105,A -85,B 0,C 180,E1 -6811.216,E2 -6811.216} C_VEL
LIN {X 0,Y 481.665,Z 126.115,A -85,B 0,C 180,E1 -6814.04,E2 -6814.04} C_VEL
LIN {X 0,Y 481.675,Z 126.104,A -85,B 0,C 180,E1 -6816.812,E2 -6816.812} C_VEL
LIN {X 0,Y 481.696,Z 126.108,A -85,B 0,C 180,E1 -6819.502,E2 -6819.502} C_VEL
LIN {X 0,Y 481.688,Z 126.108,A -85,B 0,C 180,E1 -6822.157,E2 -6822.157} C_VEL
LIN {X 0,Y 481.741,Z 126.097,A -85,B 0,C 180,E1 -6824.775,E2 -6824.775} C_VEL
LIN {X 0,Y 481.752,Z 126.098,A -85,B 0,C 180,E1 -6828.215,E2 -6828.215} C_VEL
LIN {X 0,Y 481.762,Z 126.1,A -85,B 0,C 180,E1 -6831.611,E2 -6831.611} C_VEL
LIN {X 0,Y 481.808,Z 126.088,A -85,B 0,C 180,E1 -6834.139,E2 -6834.139} C_VEL
LIN {X 0,Y 481.928,Z 126.078,A -85,B 0,C 180,E1 -6837.492,E2 -6837.492} C_VEL
LIN {X 0,Y 481.886,Z 126.082,A -85,B 0,C 180,E1 -6840.835,E2 -6840.835} C_VEL
LIN {X 0,Y 481.927,Z 126.074,A -85,B 0,C 180,E1 -6842.507,E2 -6842.507} C_VEL
LIN {X 0,Y 481.801,Z 126.092,A -85,B 0,C 180,E1 -6845.86,E2 -6845.86} C_VEL
LIN {X 0,Y 481.74,Z 126.098,A -85,B 0,C 180,E1 -6848.388,E2 -6848.388} C_VEL
LIN {X 0,Y 481.751,Z 126.096,A -85,B 0,C 180,E1 -6851.785,E2 -6851.785} C_VEL
LIN {X 0,Y 481.742,Z 126.1,A -85,B 0,C 180,E1 -6855.224,E2 -6855.224} C_VEL
LIN {X 0,Y 481.708,Z 126.109,A -85,B 0,C 180,E1 -6858.722,E2 -6858.722} C_VEL
LIN {X 0,Y 481.645,Z 126.112,A -85,B 0,C 180,E1 -6861.394,E2 -6861.394} C_VEL
LIN {X 0,Y 481.673,Z 126.107,A -85,B 0,C 180,E1 -6864.113,E2 -6864.113} C_VEL
LIN {X 0,Y 481.745,Z 126.101,A -85,B 0,C 180,E1 -6867.139,E2 -6867.139} C_VEL
LIN {X 0,Y 481.678,Z 126.105,A -85,B 0,C 180,E1 -6869.741,E2 -6869.741} C_VEL
LIN {X 0,Y 481.669,Z 126.113,A -85,B 0,C 180,E1 -6872.674,E2 -6872.674} C_VEL
LIN {X 0,Y 481.634,Z 126.112,A -85,B 0,C 180,E1 -6875.709,E2 -6875.709} C_VEL
LIN {X 0,Y 481.669,Z 126.104,A -85,B 0,C 180,E1 -6878.859,E2 -6878.859} C_VEL
LIN {X 0,Y 481.651,Z 126.114,A -85,B 0,C 180,E1 -6881.913,E2 -6881.913} C_VEL
LIN {X 0,Y 481.658,Z 126.115,A -85,B 0,C 180,E1 -6884.457,E2 -6884.457} C_VEL
LIN {X 0,Y 481.646,Z 126.112,A -85,B 0,C 180,E1 -6887.839,E2 -6887.839} C_VEL
LIN {X 0,Y 481.679,Z 126.111,A -85,B 0,C 180,E1 -6890.651,E2 -6890.651} C_VEL
LIN {X 0,Y 481.626,Z 126.114,A -85,B 0,C 180,E1 -6893.376,E2 -6893.376} C_VEL
LIN {X 0,Y 481.708,Z 126.106,A -85,B 0,C 180,E1 -6896.33,E2 -6896.33} C_VEL
LIN {X 0,Y 481.677,Z 126.112,A -85,B 0,C 180,E1 -6900.018,E2 -6900.018} C_VEL
LIN {X 0,Y 481.7,Z 126.204,A -85,B 0,C 180,E1 -6900.14,E2 -6900.14} C_VEL
LIN {X 0,Y 485.313,Z 140.84,A -85,B 0,C 180,E1 -6902.627,E2 -6902.627} C_VEL
LIN {X 0,Y 485.908,Z 145.473,A -85,B 0,C 180,E1 -6903.361,E2 -6903.361} C_VEL
LIN {X 0,Y 484.856,Z 166.038,A -85,B 0,C 180,E1 -6906.34,E2 -6906.34} C_VEL
LIN {X 0,Y 484.789,Z 167.58,A -85,B 0,C 180,E1 -6906.526,E2 -6906.526} C_VEL
LIN {X 0,Y 489.058,Z 189.02,A -85,B 0,C 180,E1 -6907.096,E2 -6907.096} C_VEL
LIN {X 0,Y 487.51,Z 333.397,A -85,B 0,C 180,E1 -6909.317,E2 -6909.317} C_VEL
LIN {X 0,Y 486.96,Z 348.758,A -85,B 0,C 180,E1 -6909.707,E2 -6909.707} C_VEL
LIN {X 0,Y 486.423,Z 363.535,A -85,B 0,C 180,E1 -6910.257,E2 -6910.257} C_VEL
LIN {X 0,Y 485.702,Z 378.609,A -85,B 0,C 180,E1 -6911,E2 -6911} C_VEL
LIN {X 0,Y 485,Z 392.092,A -85,B 0,C 180,E1 -6911.848,E2 -6911.848} C_VEL
LIN {X 0,Y 484.244,Z 404.538,A -85,B 0,C 180,E1 -6912.8,E2 -6912.8} C_VEL
LIN {X 0,Y 483.472,Z 417.207,A -85,B 0,C 180,E1 -6913.967,E2 -6913.967} C_VEL
LIN {X 0,Y 482.771,Z 428.726,A -85,B 0,C 180,E1 -6915.241,E2 -6915.241} C_VEL
LIN {X 0,Y 482.22,Z 438.437,A -85,B 0,C 180,E1 -6916.515,E2 -6916.515} C_VEL
LIN {X 0,Y 481.746,Z 447.784,A -85,B 0,C 180,E1 -6917.966,E2 -6917.966} C_VEL
LIN {X 0,Y 481.43,Z 455.95,A -85,B 0,C 180,E1 -6919.486,E2 -6919.486} C_VEL
LIN {X 0,Y 481.089,Z 463.381,A -85,B 0,C 180,E1 -6921.177,E2 -6921.177} C_VEL
LIN {X 0,Y 480.97,Z 469.281,A -85,B 0,C 180,E1 -6922.866,E2 -6922.866} C_VEL
LIN {X 0,Y 480.878,Z 472.787,A -85,B 0,C 180,E1 -6924.128,E2 -6924.128} C_VEL
LIN {X 0,Y 480.774,Z 476.331,A -85,B 0,C 180,E1 -6925.809,E2 -6925.809} C_VEL
LIN {X 0,Y 480.817,Z 478.668,A -85,B 0,C 180,E1 -6927.487,E2 -6927.487} C_VEL
LIN {X 0,Y 480.756,Z 479.844,A -85,B 0,C 180,E1 -6929.163,E2 -6929.163} C_VEL
LIN {X 0,Y 480.756,Z 479.848,A -85,B 0,C 180,E1 -6930.838,E2 -6930.838} C_VEL
LIN {X 0,Y 480.817,Z 478.677,A -85,B 0,C 180,E1 -6932.514,E2 -6932.514} C_VEL
LIN {X 0,Y 480.774,Z 476.346,A -85,B 0,C 180,E1 -6934.192,E2 -6934.192} C_VEL
LIN {X 0,Y 480.884,Z 472.811,A -85,B 0,C 180,E1 -6935.872,E2 -6935.872} C_VEL
LIN {X 0,Y 480.984,Z 467.977,A -85,B 0,C 180,E1 -6937.557,E2 -6937.557} C_VEL
LIN {X 0,Y 481.147,Z 461.713,A -85,B 0,C 180,E1 -6939.246,E2 -6939.246} C_VEL
LIN {X 0,Y 481.548,Z 453.848,A -85,B 0,C 180,E1 -6940.937,E2 -6940.937} C_VEL
LIN {X 0,Y 481.805,Z 445.992,A -85,B 0,C 180,E1 -6942.341,E2 -6942.341} C_VEL
LIN {X 0,Y 482.406,Z 435.386,A -85,B 0,C 180,E1 -6943.91,E2 -6943.91} C_VEL
LIN {X 0,Y 482.976,Z 425.08,A -85,B 0,C 180,E1 -6945.185,E2 -6945.185} C_VEL
LIN {X 0,Y 483.664,Z 414.223,A -85,B 0,C 180,E1 -6946.316,E2 -6946.316} C_VEL
LIN {X 0,Y 484.327,Z 401.708,A -85,B 0,C 180,E1 -6947.415,E2 -6947.415} C_VEL
LIN {X 0,Y 485.147,Z 388.511,A -85,B 0,C 180,E1 -6948.366,E2 -6948.366} C_VEL
LIN {X 0,Y 485.78,Z 375.985,A -85,B 0,C 180,E1 -6949.107,E2 -6949.107} C_VEL
LIN {X 0,Y 486.457,Z 361.35,A -85,B 0,C 180,E1 -6949.794,E2 -6949.794} C_VEL
LIN {X 0,Y 486.959,Z 346.303,A -85,B 0,C 180,E1 -6950.322,E2 -6950.322} C_VEL
LIN {X 0,Y 487.378,Z 330.597,A -85,B 0,C 180,E1 -6950.689,E2 -6950.689} C_VEL
LIN {X 0,Y 488.889,Z 189.924,A -85,B 0,C 180,E1 -6952.822,E2 -6952.822} C_VEL
LIN {X 0,Y 484.648,Z 167.483,A -85,B 0,C 180,E1 -6953.393,E2 -6953.393} C_VEL
LIN {X 0,Y 485.604,Z 147.802,A -85,B 0,C 180,E1 -6956.194,E2 -6956.194} C_VEL
LIN {X 0,Y 485.63,Z 143.043,A -85,B 0,C 180,E1 -6956.888,E2 -6956.888} C_VEL
LIN {X 0,Y 482.142,Z 128.024,A -85,B 0,C 180,E1 -6959.319,E2 -6959.319} C_VEL
LIN {X 0,Y 481.682,Z 126.112,A -85,B 0,C 180,E1 -6959.643,E2 -6959.643} C_VEL
LIN {X 0,Y 481.673,Z 126.113,A -85,B 0,C 180,E1 -6962.675,E2 -6962.675} C_VEL
LIN {X 0,Y 481.638,Z 126.12,A -85,B 0,C 180,E1 -6965.71,E2 -6965.71} C_VEL
LIN {X 0,Y 481.673,Z 126.108,A -85,B 0,C 180,E1 -6968.86,E2 -6968.86} C_VEL
LIN {X 0,Y 481.648,Z 126.116,A -85,B 0,C 180,E1 -6971.912,E2 -6971.912} C_VEL
LIN {X 0,Y 481.656,Z 126.112,A -85,B 0,C 180,E1 -6974.458,E2 -6974.458} C_VEL
LIN {X 0,Y 481.65,Z 126.116,A -85,B 0,C 180,E1 -6977.84,E2 -6977.84} C_VEL
LIN {X 0,Y 481.661,Z 126.107,A -85,B 0,C 180,E1 -6980.655,E2 -6980.655} C_VEL
LIN {X 0,Y 481.63,Z 126.119,A -85,B 0,C 180,E1 -6983.377,E2 -6983.377} C_VEL
LIN {X 0,Y 481.68,Z 126.106,A -85,B 0,C 180,E1 -6986.328,E2 -6986.328} C_VEL
LIN {X 0,Y 481.649,Z 126.113,A -85,B 0,C 180,E1 -6989.419,E2 -6989.419} C_VEL
LIN {X 0,Y 481.661,Z 126.098,A -85,B 0,C 180,E1 -6992.166,E2 -6992.166} C_VEL
LIN {X 0,Y 481.679,Z 126.11,A -85,B 0,C 180,E1 -6994.968,E2 -6994.968} C_VEL
LIN {X 0,Y 481.651,Z 126.107,A -85,B 0,C 180,E1 -6997.705,E2 -6997.705} C_VEL
LIN {X 0,Y 481.706,Z 126.105,A -85,B 0,C 180,E1 -7000.393,E2 -7000.393} C_VEL
LIN {X 0,Y 481.675,Z 126.108,A -85,B 0,C 180,E1 -7003.034,E2 -7003.034} C_VEL
LIN {X 0,Y 481.679,Z 126.106,A -85,B 0,C 180,E1 -7005.639,E2 -7005.639} C_VEL
LIN {X 0,Y 481.756,Z 126.097,A -85,B 0,C 180,E1 -7008.216,E2 -7008.216} C_VEL
LIN {X 0,Y 481.733,Z 126.098,A -85,B 0,C 180,E1 -7011.612,E2 -7011.612} C_VEL
LIN {X 0,Y 481.777,Z 126.097,A -85,B 0,C 180,E1 -7014.139,E2 -7014.139} C_VEL
LIN {X 0,Y 481.911,Z 126.073,A -85,B 0,C 180,E1 -7017.493,E2 -7017.493} C_VEL
LIN {X 0,Y 481.915,Z 126.067,A -85,B 0,C 180,E1 -7020,E2 -7020} C_VEL
LIN {X 0,Y 481.91,Z 126.079,A -85,B 0,C 180,E1 -7022.508,E2 -7022.508} C_VEL
LIN {X 0,Y 481.776,Z 126.099,A -85,B 0,C 180,E1 -7025.861,E2 -7025.861} C_VEL
LIN {X 0,Y 481.717,Z 126.091,A -85,B 0,C 180,E1 -7028.389,E2 -7028.389} C_VEL
LIN {X 0,Y 481.73,Z 126.098,A -85,B 0,C 180,E1 -7031.786,E2 -7031.786} C_VEL
LIN {X 0,Y 481.695,Z 126.106,A -85,B 0,C 180,E1 -7035.226,E2 -7035.226} C_VEL
LIN {X 0,Y 481.626,Z 126.112,A -85,B 0,C 180,E1 -7038.726,E2 -7038.726} C_VEL
LIN {X 0,Y 481.624,Z 126.118,A -85,B 0,C 180,E1 -7041.396,E2 -7041.396} C_VEL
LIN {X 0,Y 481.617,Z 126.115,A -85,B 0,C 180,E1 -7044.117,E2 -7044.117} C_VEL
LIN {X 0,Y 481.646,Z 126.113,A -85,B 0,C 180,E1 -7047.114,E2 -7047.114} C_VEL
LIN {X 0,Y 481.605,Z 126.107,A -85,B 0,C 180,E1 -7049.747,E2 -7049.747} C_VEL
LIN {X 0,Y 481.638,Z 126.11,A -85,B 0,C 180,E1 -7052.677,E2 -7052.677} C_VEL
LIN {X 0,Y 481.648,Z 126.113,A -85,B 0,C 180,E1 -7055.201,E2 -7055.201} C_VEL
LIN {X 0,Y 481.632,Z 126.1,A -85,B 0,C 180,E1 -7058.003,E2 -7058.003} C_VEL
LIN {X 0,Y 481.628,Z 126.119,A -85,B 0,C 180,E1 -7061.045,E2 -7061.045} C_VEL
LIN {X 0,Y 481.659,Z 126.11,A -85,B 0,C 180,E1 -7064.458,E2 -7064.458} C_VEL
LIN {X 0,Y 481.62,Z 126.114,A -85,B 0,C 180,E1 -7066.855,E2 -7066.855} C_VEL
LIN {X 0,Y 481.661,Z 126.11,A -85,B 0,C 180,E1 -7070.057,E2 -7070.057} C_VEL
LIN {X 0,Y 481.626,Z 126.111,A -85,B 0,C 180,E1 -7073.377,E2 -7073.377} C_VEL
LIN {X 0,Y 481.676,Z 126.112,A -85,B 0,C 180,E1 -7076.327,E2 -7076.327} C_VEL
LIN {X 0,Y 481.651,Z 126.111,A -85,B 0,C 180,E1 -7079.418,E2 -7079.418} C_VEL
LIN {X 0,Y 481.656,Z 126.113,A -85,B 0,C 180,E1 -7082.165,E2 -7082.165} C_VEL
LIN {X 0,Y 481.679,Z 126.108,A -85,B 0,C 180,E1 -7084.967,E2 -7084.967} C_VEL
LIN {X 0,Y 481.641,Z 126.114,A -85,B 0,C 180,E1 -7087.938,E2 -7087.938} C_VEL
LIN {X 0,Y 480.973,Z 126.197,A -85,B 0,C 180,E1 -7088.636,E2 -7088.636} C_VEL
LIN {X 0,Y 478.15,Z 126.551,A -85,B 0,C 180,E1 -7089.77,E2 -7089.77} C_VEL
LIN {X 0,Y 475.765,Z 126.846,A -85,B 0,C 180,E1 -7090.684,E2 -7090.684} C_VEL
LIN {X 0,Y 474.736,Z 126.971,A -85,B 0,C 180,E1 -7091.39,E2 -7091.39} C_VEL
LIN {X 0,Y 474.65,Z 126.98,A -85,B 0,C 180,E1 -7091.629,E2 -7091.629} C_VEL
LIN {X 0,Y 474.704,Z 126.977,A -85,B 0,C 180,E1 -7094.544,E2 -7094.544} C_VEL
LIN {X 0,Y 474.71,Z 126.98,A -85,B 0,C 180,E1 -7098.037,E2 -7098.037} C_VEL
LIN {X 0,Y 474.714,Z 126.981,A -85,B 0,C 180,E1 -7101.486,E2 -7101.486} C_VEL
LIN {X 0,Y 474.746,Z 127.111,A -85,B 0,C 180,E1 -7102.399,E2 -7102.399} C_VEL
LIN {X 0,Y 477.572,Z 139.785,A -85,B 0,C 180,E1 -7104.722,E2 -7104.722} C_VEL
LIN {X 0,Y 478.025,Z 143.439,A -85,B 0,C 180,E1 -7105.361,E2 -7105.361} C_VEL
LIN {X 0,Y 482.444,Z 163.537,A -85,B 0,C 180,E1 -7105.902,E2 -7105.902} C_VEL
LIN {X 0,Y 480.832,Z 308.34,A -85,B 0,C 180,E1 -7108.141,E2 -7108.141} C_VEL
LIN {X 0,Y 480.459,Z 323.285,A -85,B 0,C 180,E1 -7108.533,E2 -7108.533} C_VEL
LIN {X 0,Y 479.9,Z 338.526,A -85,B 0,C 180,E1 -7109.108,E2 -7109.108} C_VEL
LIN {X 0,Y 479.275,Z 352.123,A -85,B 0,C 180,E1 -7109.79,E2 -7109.79} C_VEL
LIN {X 0,Y 478.554,Z 365.287,A -85,B 0,C 180,E1 -7110.613,E2 -7110.613} C_VEL
LIN {X 0,Y 477.762,Z 378.005,A -85,B 0,C 180,E1 -7111.585,E2 -7111.585} C_VEL
LIN {X 0,Y 476.96,Z 390.538,A -85,B 0,C 180,E1 -7112.745,E2 -7112.745} C_VEL
LIN {X 0,Y 476.228,Z 401.991,A -85,B 0,C 180,E1 -7114.019,E2 -7114.019} C_VEL
LIN {X 0,Y 475.612,Z 411.677,A -85,B 0,C 180,E1 -7115.299,E2 -7115.299} C_VEL
LIN {X 0,Y 475.046,Z 421.2,A -85,B 0,C 180,E1 -7116.797,E2 -7116.797} C_VEL
LIN {X 0,Y 474.632,Z 429.164,A -85,B 0,C 180,E1 -7118.301,E2 -7118.301} C_VEL
LIN {X 0,Y 474.25,Z 435.827,A -85,B 0,C 180,E1 -7119.812,E2 -7119.812} C_VEL
LIN {X 0,Y 474.018,Z 441.739,A -85,B 0,C 180,E1 -7121.481,E2 -7121.481} C_VEL
LIN {X 0,Y 473.839,Z 446.67,A -85,B 0,C 180,E1 -7123.291,E2 -7123.291} C_VEL
LIN {X 0,Y 473.686,Z 450.541,A -85,B 0,C 180,E1 -7125.333,E2 -7125.333} C_VEL
LIN {X 0,Y 473.627,Z 452.633,A -85,B 0,C 180,E1 -7127.264,E2 -7127.264} C_VEL
LIN {X 0,Y 473.613,Z 453.28,A -85,B 0,C 180,E1 -7129.054,E2 -7129.054} C_VEL
LIN {X 0,Y 473.651,Z 452.639,A -85,B 0,C 180,E1 -7130.861,E2 -7130.861} C_VEL
LIN {X 0,Y 473.677,Z 450.685,A -85,B 0,C 180,E1 -7132.691,E2 -7132.691} C_VEL
LIN {X 0,Y 473.848,Z 447.336,A -85,B 0,C 180,E1 -7134.537,E2 -7134.537} C_VEL
LIN {X 0,Y 474.009,Z 442.461,A -85,B 0,C 180,E1 -7136.41,E2 -7136.41} C_VEL
LIN {X 0,Y 474.203,Z 437.668,A -85,B 0,C 180,E1 -7137.83,E2 -7137.83} C_VEL
LIN {X 0,Y 474.534,Z 430.744,A -85,B 0,C 180,E1 -7139.501,E2 -7139.501} C_VEL
LIN {X 0,Y 475.061,Z 422.125,A -85,B 0,C 180,E1 -7141.184,E2 -7141.184} C_VEL
LIN {X 0,Y 475.603,Z 413.275,A -85,B 0,C 180,E1 -7142.616,E2 -7142.616} C_VEL
LIN {X 0,Y 476.266,Z 403.257,A -85,B 0,C 180,E1 -7143.98,E2 -7143.98} C_VEL
LIN {X 0,Y 476.962,Z 392.592,A -85,B 0,C 180,E1 -7145.205,E2 -7145.205} C_VEL
LIN {X 0,Y 477.844,Z 379.754,A -85,B 0,C 180,E1 -7146.429,E2 -7146.429} C_VEL
LIN {X 0,Y 478.631,Z 366.85,A -85,B 0,C 180,E1 -7147.446,E2 -7147.446} C_VEL
LIN {X 0,Y 479.434,Z 352.96,A -85,B 0,C 180,E1 -7148.335,E2 -7148.335} C_VEL
LIN {X 0,Y 480.116,Z 338.099,A -85,B 0,C 180,E1 -7149.083,E2 -7149.083} C_VEL
LIN {X 0,Y 480.634,Z 322.482,A -85,B 0,C 180,E1 -7149.669,E2 -7149.669} C_VEL
LIN {X 0,Y 481.083,Z 307.564,A -85,B 0,C 180,E1 -7150.049,E2 -7150.049} C_VEL
LIN {X 0,Y 482.841,Z 163.132,A -85,B 0,C 180,E1 -7152.303,E2 -7152.303} C_VEL
LIN {X 0,Y 478.251,Z 143.712,A -85,B 0,C 180,E1 -7152.887,E2 -7152.887} C_VEL
LIN {X 0,Y 476.108,Z 133.071,A -85,B 0,C 180,E1 -7154.883,E2 -7154.883} C_VEL
LIN {X 0,Y 474.62,Z 126.992,A -85,B 0,C 180,E1 -7156.071,E2 -7156.071} C_VEL
LIN {X 0,Y 474.616,Z 126.994,A -85,B 0,C 180,E1 -7159.341,E2 -7159.341} C_VEL
LIN {X 0,Y 474.586,Z 126.994,A -85,B 0,C 180,E1 -7162.615,E2 -7162.615} C_VEL
LIN {X 0,Y 474.633,Z 126.983,A -85,B 0,C 180,E1 -7165.758,E2 -7165.758} C_VEL
LIN {X 0,Y 474.599,Z 126.99,A -85,B 0,C 180,E1 -7168.782,E2 -7168.782} C_VEL
LIN {X 0,Y 474.621,Z 126.983,A -85,B 0,C 180,E1 -7171.715,E2 -7171.715} C_VEL
LIN {X 0,Y 474.629,Z 126.984,A -85,B 0,C 180,E1 -7174.588,E2 -7174.588} C_VEL
LIN {X 0,Y 474.601,Z 126.986,A -85,B 0,C 180,E1 -7177.355,E2 -7177.355} C_VEL
LIN {X 0,Y 474.654,Z 126.987,A -85,B 0,C 180,E1 -7180.089,E2 -7180.089} C_VEL
LIN {X 0,Y 474.634,Z 126.983,A -85,B 0,C 180,E1 -7182.773,E2 -7182.773} C_VEL
LIN {X 0,Y 474.643,Z 126.984,A -85,B 0,C 180,E1 -7185.42,E2 -7185.42} C_VEL
LIN {X 0,Y 474.705,Z 126.977,A -85,B 0,C 180,E1 -7188.037,E2 -7188.037} C_VEL
LIN {X 0,Y 474.727,Z 126.975,A -85,B 0,C 180,E1 -7191.486,E2 -7191.486} C_VEL
LIN {X 0,Y 474.77,Z 126.965,A -85,B 0,C 180,E1 -7194.052,E2 -7194.052} C_VEL
LIN {X 0,Y 474.894,Z 126.955,A -85,B 0,C 180,E1 -7197.455,E2 -7197.455} C_VEL
LIN {X 0,Y 474.912,Z 126.951,A -85,B 0,C 180,E1 -7200,E2 -7200} C_VEL
LIN {X 0,Y 474.893,Z 126.95,A -85,B 0,C 180,E1 -7202.544,E2 -7202.544} C_VEL
LIN {X 0,Y 474.762,Z 126.968,A -85,B 0,C 180,E1 -7205.947,E2 -7205.947} C_VEL
LIN {X 0,Y 474.711,Z 126.974,A -85,B 0,C 180,E1 -7208.513,E2 -7208.513} C_VEL
LIN {X 0,Y 474.704,Z 126.973,A -85,B 0,C 180,E1 -7211.962,E2 -7211.962} C_VEL
LIN {X 0,Y 474.699,Z 126.975,A -85,B 0,C 180,E1 -7215.455,E2 -7215.455} C_VEL
LIN {X 0,Y 474.662,Z 126.983,A -85,B 0,C 180,E1 -7219.01,E2 -7219.01} C_VEL
LIN {X 0,Y 474.588,Z 126.99,A -85,B 0,C 180,E1 -7221.729,E2 -7221.729} C_VEL
LIN {X 0,Y 474.654,Z 126.985,A -85,B 0,C 180,E1 -7224.493,E2 -7224.493} C_VEL
LIN {X 0,Y 474.68,Z 126.98,A -85,B 0,C 180,E1 -7227.334,E2 -7227.334} C_VEL
LIN {X 0,Y 474.603,Z 126.993,A -85,B 0,C 180,E1 -7230.81,E2 -7230.81} C_VEL
LIN {X 0,Y 474.623,Z 126.987,A -85,B 0,C 180,E1 -7233.221,E2 -7233.221} C_VEL
LIN {X 0,Y 474.587,Z 126.996,A -85,B 0,C 180,E1 -7236.323,E2 -7236.323} C_VEL
LIN {X 0,Y 474.616,Z 126.982,A -85,B 0,C 180,E1 -7239.646,E2 -7239.646} C_VEL
LIN {X 0,Y 474.613,Z 126.981,A -85,B 0,C 180,E1 -7242.934,E2 -7242.934} C_VEL
LIN {X 0,Y 474.608,Z 126.992,A -85,B 0,C 180,E1 -7245.895,E2 -7245.895} C_VEL
LIN {X 0,Y 474.626,Z 126.986,A -85,B 0,C 180,E1 -7249.041,E2 -7249.041} C_VEL
LIN {X 0,Y 474.609,Z 126.993,A -85,B 0,C 180,E1 -7251.704,E2 -7251.704} C_VEL
LIN {X 0,Y 474.623,Z 126.985,A -85,B 0,C 180,E1 -7254.726,E2 -7254.726} C_VEL
LIN {X 0,Y 474.634,Z 126.989,A -85,B 0,C 180,E1 -7257.788,E2 -7257.788} C_VEL
LIN {X 0,Y 474.649,Z 127.027,A -85,B 0,C 180,E1 -7259.773,E2 -7259.773} C_VEL
LIN {X 0,Y 478.472,Z 142.47,A -85,B 0,C 180,E1 -7262.452,E2 -7262.452} C_VEL
LIN {X 0,Y 479.135,Z 146.789,A -85,B 0,C 180,E1 -7263.154,E2 -7263.154} C_VEL
LIN {X 0,Y 478.042,Z 167.041,A -85,B 0,C 180,E1 -7266.141,E2 -7266.141} C_VEL
LIN {X 0,Y 482.596,Z 191.111,A -85,B 0,C 180,E1 -7266.79,E2 -7266.79} C_VEL
LIN {X 0,Y 480.884,Z 333.83,A -85,B 0,C 180,E1 -7269.019,E2 -7269.019} C_VEL
LIN {X 0,Y 480.294,Z 349.732,A -85,B 0,C 180,E1 -7269.44,E2 -7269.44} C_VEL
LIN {X 0,Y 479.73,Z 363.919,A -85,B 0,C 180,E1 -7269.985,E2 -7269.985} C_VEL
LIN {X 0,Y 478.967,Z 378.572,A -85,B 0,C 180,E1 -7270.722,E2 -7270.722} C_VEL
LIN {X 0,Y 478.208,Z 392.023,A -85,B 0,C 180,E1 -7271.581,E2 -7271.581} C_VEL
LIN {X 0,Y 477.328,Z 405.738,A -85,B 0,C 180,E1 -7272.654,E2 -7272.654} C_VEL
LIN {X 0,Y 476.516,Z 418.168,A -85,B 0,C 180,E1 -7273.837,E2 -7273.837} C_VEL
LIN {X 0,Y 475.744,Z 430.369,A -85,B 0,C 180,E1 -7275.237,E2 -7275.237} C_VEL
LIN {X 0,Y 475.059,Z 441.228,A -85,B 0,C 180,E1 -7276.744,E2 -7276.744} C_VEL
LIN {X 0,Y 474.592,Z 450.28,A -85,B 0,C 180,E1 -7278.252,E2 -7278.252} C_VEL
LIN {X 0,Y 474.238,Z 457.792,A -85,B 0,C 180,E1 -7279.757,E2 -7279.757} C_VEL
LIN {X 0,Y 473.972,Z 464.814,A -85,B 0,C 180,E1 -7281.473,E2 -7281.473} C_VEL
LIN {X 0,Y 473.828,Z 470.341,A -85,B 0,C 180,E1 -7283.186,E2 -7283.186} C_VEL
LIN {X 0,Y 473.778,Z 474.521,A -85,B 0,C 180,E1 -7284.894,E2 -7284.894} C_VEL
LIN {X 0,Y 473.739,Z 477.452,A -85,B 0,C 180,E1 -7286.598,E2 -7286.598} C_VEL
LIN {X 0,Y 473.695,Z 479.201,A -85,B 0,C 180,E1 -7288.3,E2 -7288.3} C_VEL
LIN {X 0,Y 473.667,Z 479.802,A -85,B 0,C 180,E1 -7290,E2 -7290} C_VEL
LIN {X 0,Y 473.695,Z 479.205,A -85,B 0,C 180,E1 -7291.701,E2 -7291.701} C_VEL
LIN {X 0,Y 473.739,Z 477.456,A -85,B 0,C 180,E1 -7293.402,E2 -7293.402} C_VEL
LIN {X 0,Y 473.779,Z 474.528,A -85,B 0,C 180,E1 -7295.107,E2 -7295.107} C_VEL
LIN {X 0,Y 473.887,Z 470.353,A -85,B 0,C 180,E1 -7296.814,E2 -7296.814} C_VEL
LIN {X 0,Y 473.977,Z 464.815,A -85,B 0,C 180,E1 -7298.527,E2 -7298.527} C_VEL
LIN {X 0,Y 474.243,Z 457.77,A -85,B 0,C 180,E1 -7300.244,E2 -7300.244} C_VEL
LIN {X 0,Y 474.615,Z 450.236,A -85,B 0,C 180,E1 -7301.748,E2 -7301.748} C_VEL
LIN {X 0,Y 475.052,Z 441.137,A -85,B 0,C 180,E1 -7303.257,E2 -7303.257} C_VEL
LIN {X 0,Y 475.718,Z 430.179,A -85,B 0,C 180,E1 -7304.765,E2 -7304.765} C_VEL
LIN {X 0,Y 476.434,Z 418.9,A -85,B 0,C 180,E1 -7306.057,E2 -7306.057} C_VEL
LIN {X 0,Y 477.19,Z 406.522,A -85,B 0,C 180,E1 -7307.242,E2 -7307.242} C_VEL
LIN {X 0,Y 478.074,Z 392.878,A -85,B 0,C 180,E1 -7308.315,E2 -7308.315} C_VEL
LIN {X 0,Y 478.801,Z 379.462,A -85,B 0,C 180,E1 -7309.174,E2 -7309.174} C_VEL
LIN {X 0,Y 479.593,Z 364.25,A -85,B 0,C 180,E1 -7309.942,E2 -7309.942} C_VEL
LIN {X 0,Y 480.185,Z 348.734,A -85,B 0,C 180,E1 -7310.527,E2 -7310.527} C_VEL
LIN {X 0,Y 480.639,Z 332.639,A -85,B 0,C 180,E1 -7310.937,E2 -7310.937} C_VEL
LIN {X 0,Y 482.296,Z 190.688,A -85,B 0,C 180,E1 -7313.121,E2 -7313.121} C_VEL
LIN {X 0,Y 477.846,Z 167.273,A -85,B 0,C 180,E1 -7313.731,E2 -7313.731} C_VEL
LIN {X 0,Y 478.804,Z 148.483,A -85,B 0,C 180,E1 -7316.444,E2 -7316.444} C_VEL
LIN {X 0,Y 478.689,Z 144.292,A -85,B 0,C 180,E1 -7317.074,E2 -7317.074} C_VEL
LIN {X 0,Y 475.321,Z 129.818,A -85,B 0,C 180,E1 -7319.448,E2 -7319.448} C_VEL
LIN {X 0,Y 474.639,Z 126.988,A -85,B 0,C 180,E1 -7319.952,E2 -7319.952} C_VEL
LIN {X 0,Y 474.644,Z 126.988,A -85,B 0,C 180,E1 -7323.22,E2 -7323.22} C_VEL
LIN {X 0,Y 474.591,Z 126.996,A -85,B 0,C 180,E1 -7326.324,E2 -7326.324} C_VEL
LIN {X 0,Y 474.615,Z 126.994,A -85,B 0,C 180,E1 -7329.646,E2 -7329.646} C_VEL
LIN {X 0,Y 474.602,Z 126.99,A -85,B 0,C 180,E1 -7332.234,E2 -7332.234} C_VEL
LIN {X 0,Y 474.619,Z 126.992,A -85,B 0,C 180,E1 -7335.298,E2 -7335.298} C_VEL
LIN {X 0,Y 474.623,Z 126.988,A -85,B 0,C 180,E1 -7338.215,E2 -7338.215} C_VEL
LIN {X 0,Y 474.613,Z 126.99,A -85,B 0,C 180,E1 -7341.543,E2 -7341.543} C_VEL
LIN {X 0,Y 474.625,Z 126.985,A -85,B 0,C 180,E1 -7344.726,E2 -7344.726} C_VEL
LIN {X 0,Y 474.638,Z 126.984,A -85,B 0,C 180,E1 -7347.788,E2 -7347.788} C_VEL
LIN {X 0,Y 474.602,Z 126.99,A -85,B 0,C 180,E1 -7350.891,E2 -7350.891} C_VEL
LIN {X 0,Y 474.616,Z 126.982,A -85,B 0,C 180,E1 -7353.626,E2 -7353.626} C_VEL
LIN {X 0,Y 474.638,Z 126.987,A -85,B 0,C 180,E1 -7356.642,E2 -7356.642} C_VEL
LIN {X 0,Y 474.656,Z 126.981,A -85,B 0,C 180,E1 -7360.09,E2 -7360.09} C_VEL
LIN {X 0,Y 474.636,Z 126.986,A -85,B 0,C 180,E1 -7362.774,E2 -7362.774} C_VEL
LIN {X 0,Y 474.64,Z 126.983,A -85,B 0,C 180,E1 -7365.421,E2 -7365.421} C_VEL
LIN {X 0,Y 474.709,Z 126.973,A -85,B 0,C 180,E1 -7368.038,E2 -7368.038} C_VEL
LIN {X 0,Y 474.708,Z 126.973,A -85,B 0,C 180,E1 -7371.486,E2 -7371.486} C_VEL
LIN {X 0,Y 474.741,Z 126.973,A -85,B 0,C 180,E1 -7374.052,E2 -7374.052} C_VEL
LIN {X 0,Y 474.876,Z 126.949,A -85,B 0,C 180,E1 -7377.456,E2 -7377.456} C_VEL
LIN {X 0,Y 474.884,Z 126.942,A -85,B 0,C 180,E1 -7380,E2 -7380} C_VEL
LIN {X 0,Y 474.875,Z 126.954,A -85,B 0,C 180,E1 -7382.545,E2 -7382.545} C_VEL
LIN {X 0,Y 474.74,Z 126.975,A -85,B 0,C 180,E1 -7385.948,E2 -7385.948} C_VEL
LIN {X 0,Y 474.665,Z 126.967,A -85,B 0,C 180,E1 -7388.515,E2 -7388.515} C_VEL
LIN {X 0,Y 474.689,Z 126.978,A -85,B 0,C 180,E1 -7391.963,E2 -7391.963} C_VEL
LIN {X 0,Y 474.655,Z 126.985,A -85,B 0,C 180,E1 -7395.458,E2 -7395.458} C_VEL
LIN {X 0,Y 474.583,Z 126.99,A -85,B 0,C 180,E1 -7399.014,E2 -7399.014} C_VEL
LIN {X 0,Y 474.573,Z 126.993,A -85,B 0,C 180,E1 -7401.73,E2 -7401.73} C_VEL
LIN {X 0,Y 474.584,Z 126.99,A -85,B 0,C 180,E1 -7404.497,E2 -7404.497} C_VEL
LIN {X 0,Y 474.598,Z 126.987,A -85,B 0,C 180,E1 -7407.327,E2 -7407.327} C_VEL
LIN {X 0,Y 474.554,Z 126.983,A -85,B 0,C 180,E1 -7410.234,E2 -7410.234} C_VEL
LIN {X 0,Y 474.613,Z 126.993,A -85,B 0,C 180,E1 -7413.223,E2 -7413.223} C_VEL
LIN {X 0,Y 474.572,Z 126.988,A -85,B 0,C 180,E1 -7416.326,E2 -7416.326} C_VEL
LIN {X 0,Y 474.604,Z 126.984,A -85,B 0,C 180,E1 -7419.643,E2 -7419.643} C_VEL
LIN {X 0,Y 474.581,Z 126.991,A -85,B 0,C 180,E1 -7422.23,E2 -7422.23} C_VEL
LIN {X 0,Y 474.621,Z 126.977,A -85,B 0,C 180,E1 -7425.298,E2 -7425.298} C_VEL
LIN {X 0,Y 474.597,Z 126.989,A -85,B 0,C 180,E1 -7428.211,E2 -7428.211} C_VEL
LIN {X 0,Y 474.624,Z 126.991,A -85,B 0,C 180,E1 -7430.451,E2 -7430.451} C_VEL
LIN {X 0,Y 474.588,Z 126.987,A -85,B 0,C 180,E1 -7433.676,E2 -7433.676} C_VEL
LIN {X 0,Y 474.62,Z 126.983,A -85,B 0,C 180,E1 -7436.778,E2 -7436.778} C_VEL
LIN {X 0,Y 474.603,Z 126.991,A -85,B 0,C 180,E1 -7439.769,E2 -7439.769} C_VEL
LIN {X 0,Y 474.607,Z 126.992,A -85,B 0,C 180,E1 -7442.684,E2 -7442.684} C_VEL
LIN {X 0,Y 474.632,Z 126.987,A -85,B 0,C 180,E1 -7445.505,E2 -7445.505} C_VEL
LIN {X 0,Y 474.64,Z 126.984,A -85,B 0,C 180,E1 -7448.884,E2 -7448.884} C_VEL
LIN {X 0,Y 474.65,Z 126.98,A -85,B 0,C 180,E1 -7451.629,E2 -7451.629} C_VEL
LIN {X 0,Y 473.977,Z 127.063,A -85,B 0,C 180,E1 -7452.338,E2 -7452.338} C_VEL
LIN {X 0,Y 471.131,Z 127.422,A -85,B 0,C 180,E1 -7453.489,E2 -7453.489} C_VEL
LIN {X 0,Y 468.725,Z 127.725,A -85,B 0,C 180,E1 -7454.418,E2 -7454.418} C_VEL
LIN {X 0,Y 467.686,Z 127.852,A -85,B 0,C 180,E1 -7455.135,E2 -7455.135} C_VEL
LIN {X 0,Y 467.598,Z 127.861,A -85,B 0,C 180,E1 -7455.378,E2 -7455.378} C_VEL
LIN {X 0,Y 467.656,Z 127.857,A -85,B 0,C 180,E1 -7458.734,E2 -7458.734} C_VEL
LIN {X 0,Y 467.717,Z 128.005,A -85,B 0,C 180,E1 -7462.119,E2 -7462.119} C_VEL
LIN {X 0,Y 470.737,Z 141.568,A -85,B 0,C 180,E1 -7464.646,E2 -7464.646} C_VEL
LIN {X 0,Y 471.162,Z 143.769,A -85,B 0,C 180,E1 -7465.023,E2 -7465.023} C_VEL
LIN {X 0,Y 475.803,Z 163.6,A -85,B 0,C 180,E1 -7465.578,E2 -7465.578} C_VEL
LIN {X 0,Y 474.161,Z 308.411,A -85,B 0,C 180,E1 -7467.85,E2 -7467.85} C_VEL
LIN {X 0,Y 473.713,Z 324.291,A -85,B 0,C 180,E1 -7468.273,E2 -7468.273} C_VEL
LIN {X 0,Y 473.138,Z 339.854,A -85,B 0,C 180,E1 -7468.883,E2 -7468.883} C_VEL
LIN {X 0,Y 472.499,Z 353.282,A -85,B 0,C 180,E1 -7469.574,E2 -7469.574} C_VEL
LIN {X 0,Y 471.715,Z 366.539,A -85,B 0,C 180,E1 -7470.426,E2 -7470.426} C_VEL
LIN {X 0,Y 470.862,Z 379.961,A -85,B 0,C 180,E1 -7471.488,E2 -7471.488} C_VEL
LIN {X 0,Y 470.004,Z 392.33,A -85,B 0,C 180,E1 -7472.678,E2 -7472.678} C_VEL
LIN {X 0,Y 469.291,Z 402.647,A -85,B 0,C 180,E1 -7473.864,E2 -7473.864} C_VEL
LIN {X 0,Y 468.621,Z 412.264,A -85,B 0,C 180,E1 -7475.162,E2 -7475.162} C_VEL
LIN {X 0,Y 468.047,Z 421.716,A -85,B 0,C 180,E1 -7476.682,E2 -7476.682} C_VEL
LIN {X 0,Y 467.608,Z 429.623,A -85,B 0,C 180,E1 -7478.209,E2 -7478.209} C_VEL
LIN {X 0,Y 467.137,Z 437.058,A -85,B 0,C 180,E1 -7479.963,E2 -7479.963} C_VEL
LIN {X 0,Y 466.948,Z 441.628,A -85,B 0,C 180,E1 -7481.283,E2 -7481.283} C_VEL
